LIN {X 0,Y 536.075,Z 1142.953,A -85,B 0,C 180,E1 24176.996,E2 24176.996} C_VEL
LIN {X 0,Y 540.442,Z 1123.188,A -85,B 0,C 180,E1 24174.545,E2 24174.545} C_VEL
LIN {X 0,Y 544.196,Z 1106.391,A -85,B 0,C 180,E1 24172.711,E2 24172.711} C_VEL
LIN {X 0,Y 547.982,Z 1089.375,A -85,B 0,C 180,E1 24171.05,E2 24171.05} C_VEL
LIN {X 0,Y 552.645,Z 1068.2,A -85,B 0,C 180,E1 24169.217,E2 24169.217} C_VEL
LIN {X 0,Y 557.206,Z 1046.015,A -85,B 0,C 180,E1 24167.564,E2 24167.564} C_VEL
LIN {X 0,Y 560.932,Z 1026.823,A -85,B 0,C 180,E1 24166.308,E2 24166.308} C_VEL
LIN {X 0,Y 564.507,Z 1007.094,A -85,B 0,C 180,E1 24165.17,E2 24165.17} C_VEL
LIN {X 0,Y 568.089,Z 985.711,A -85,B 0,C 180,E1 24164.098,E2 24164.098} C_VEL
LIN {X 0,Y 572.065,Z 959.057,A -85,B 0,C 180,E1 24162.974,E2 24162.974} C_VEL
LIN {X 0,Y 575.027,Z 935.232,A -85,B 0,C 180,E1 24162.158,E2 24162.158} C_VEL
LIN {X 0,Y 577.283,Z 914.135,A -85,B 0,C 180,E1 24161.567,E2 24161.567} C_VEL
LIN {X 0,Y 579.127,Z 892.797,A -85,B 0,C 180,E1 24161.086,E2 24161.086} C_VEL
LIN {X 0,Y 580.665,Z 868.419,A -85,B 0,C 180,E1 24160.665,E2 24160.665} C_VEL
LIN {X 0,Y 589.019,Z 647.142,A -85,B 0,C 180,E1 24157.424,E2 24157.424} C_VEL
LIN {X 0,Y 594.591,Z 507.254,A -85,B 0,C 180,E1 24155.344,E2 24155.344} C_VEL
LIN {X 0,Y 582.445,Z 490.253,A -85,B 0,C 180,E1 24153.234,E2 24153.234} C_VEL
LIN {X 0,Y 571.046,Z 475.195,A -85,B 0,C 180,E1 24151.071,E2 24151.071} C_VEL
LIN {X 0,Y 561.909,Z 463.769,A -85,B 0,C 180,E1 24149.181,E2 24149.181} C_VEL
LIN {X 0,Y 557.694,Z 458.589,A -85,B 0,C 180,E1 24148.251,E2 24148.251} C_VEL
LIN {X 0,Y 553.263,Z 453.23,A -85,B 0,C 180,E1 24147.227,E2 24147.227} C_VEL
LIN {X 0,Y 549.468,Z 448.48,A -85,B 0,C 180,E1 24146.302,E2 24146.302} C_VEL
LIN {X 0,Y 545.143,Z 443.711,A -85,B 0,C 180,E1 24145.213,E2 24145.213} C_VEL
LIN {X 0,Y 543.778,Z 441.838,A -85,B 0,C 180,E1 24144.845,E2 24144.845} C_VEL
LIN {X 0,Y 540.283,Z 438.305,A -85,B 0,C 180,E1 24143.91,E2 24143.91} C_VEL
LIN {X 0,Y 538.579,Z 435.768,A -85,B 0,C 180,E1 24143.41,E2 24143.41} C_VEL
LIN {X 0,Y 535.319,Z 432.979,A -85,B 0,C 180,E1 24142.485,E2 24142.485} C_VEL
LIN {X 0,Y 533.198,Z 429.458,A -85,B 0,C 180,E1 24141.796,E2 24141.796} C_VEL
LIN {X 0,Y 529.875,Z 427.069,A -85,B 0,C 180,E1 24140.779,E2 24140.779} C_VEL
LIN {X 0,Y 527.916,Z 423.816,A -85,B 0,C 180,E1 24140.078,E2 24140.078} C_VEL
LIN {X 0,Y 527.596,Z 422.918,A -85,B 0,C 180,E1 24139.946,E2 24139.946} C_VEL
LIN {X 0,Y 524.201,Z 421.053,A -85,B 0,C 180,E1 24138.806,E2 24138.806} C_VEL
LIN {X 0,Y 522.262,Z 418.242,A -85,B 0,C 180,E1 24138.04,E2 24138.04} C_VEL
LIN {X 0,Y 521.746,Z 416.24,A -85,B 0,C 180,E1 24137.731,E2 24137.731} C_VEL
LIN {X 0,Y 521.74,Z 416.177,A -85,B 0,C 180,E1 24134.2,E2 24134.2} C_VEL
LIN {X 0,Y 521.724,Z 416.212,A -85,B 0,C 180,E1 24130.826,E2 24130.826} C_VEL
LIN {X 0,Y 521.748,Z 416.194,A -85,B 0,C 180,E1 24127.267,E2 24127.267} C_VEL
LIN {X 0,Y 521.735,Z 416.182,A -85,B 0,C 180,E1 24123.846,E2 24123.846} C_VEL
LIN {X 0,Y 521.719,Z 416.225,A -85,B 0,C 180,E1 24120.439,E2 24120.439} C_VEL
LIN {X 0,Y 521.735,Z 416.172,A -85,B 0,C 180,E1 24117.034,E2 24117.034} C_VEL
LIN {X 0,Y 521.747,Z 416.238,A -85,B 0,C 180,E1 24113.508,E2 24113.508} C_VEL
LIN {X 0,Y 521.712,Z 416.179,A -85,B 0,C 180,E1 24110.067,E2 24110.067} C_VEL
LIN {X 0,Y 521.743,Z 416.199,A -85,B 0,C 180,E1 24106.592,E2 24106.592} C_VEL
LIN {X 0,Y 521.742,Z 416.215,A -85,B 0,C 180,E1 24103.064,E2 24103.064} C_VEL
LIN {X 0,Y 521.793,Z 416.552,A -85,B 0,C 180,E1 24102.836,E2 24102.836} C_VEL
LIN {X 0,Y 522.41,Z 418.598,A -85,B 0,C 180,E1 24102.311,E2 24102.311} C_VEL
LIN {X 0,Y 524.376,Z 421.238,A -85,B 0,C 180,E1 24101.547,E2 24101.547} C_VEL
LIN {X 0,Y 526.706,Z 422.973,A -85,B 0,C 180,E1 24100.741,E2 24100.741} C_VEL
LIN {X 0,Y 530.704,Z 427.887,A -85,B 0,C 180,E1 24099.37,E2 24099.37} C_VEL
LIN {X 0,Y 532.055,Z 429.416,A -85,B 0,C 180,E1 24098.936,E2 24098.936} C_VEL
LIN {X 0,Y 535.394,Z 433.498,A -85,B 0,C 180,E1 24097.894,E2 24097.894} C_VEL
LIN {X 0,Y 536.844,Z 435.07,A -85,B 0,C 180,E1 24097.467,E2 24097.467} C_VEL
LIN {X 0,Y 540.381,Z 439.58,A -85,B 0,C 180,E1 24096.442,E2 24096.442} C_VEL
LIN {X 0,Y 542.443,Z 442.092,A -85,B 0,C 180,E1 24095.873,E2 24095.873} C_VEL
LIN {X 0,Y 550.326,Z 451.99,A -85,B 0,C 180,E1 24093.832,E2 24093.832} C_VEL
LIN {X 0,Y 559.201,Z 463.612,A -85,B 0,C 180,E1 24091.745,E2 24091.745} C_VEL
LIN {X 0,Y 566.986,Z 474.312,A -85,B 0,C 180,E1 24090.061,E2 24090.061} C_VEL
LIN {X 0,Y 576.321,Z 487.386,A -85,B 0,C 180,E1 24088.197,E2 24088.197} C_VEL
LIN {X 0,Y 587.425,Z 503.948,A -85,B 0,C 180,E1 24086.149,E2 24086.149} C_VEL
LIN {X 0,Y 594.763,Z 515.576,A -85,B 0,C 180,E1 24084.879,E2 24084.879} C_VEL
LIN {X 0,Y 586.116,Z 737.329,A -85,B 0,C 180,E1 24081.599,E2 24081.599} C_VEL
LIN {X 0,Y 579.945,Z 901.421,A -85,B 0,C 180,E1 24079.193,E2 24079.193} C_VEL
LIN {X 0,Y 578.109,Z 926.813,A -85,B 0,C 180,E1 24078.724,E2 24078.724} C_VEL
LIN {X 0,Y 575.284,Z 954.698,A -85,B 0,C 180,E1 24078.019,E2 24078.019} C_VEL
LIN {X 0,Y 572.619,Z 976.547,A -85,B 0,C 180,E1 24077.322,E2 24077.322} C_VEL
LIN {X 0,Y 569.746,Z 997.313,A -85,B 0,C 180,E1 24076.532,E2 24076.532} C_VEL
LIN {X 0,Y 566.591,Z 1017.778,A -85,B 0,C 180,E1 24075.624,E2 24075.624} C_VEL
LIN {X 0,Y 562.4,Z 1042.853,A -85,B 0,C 180,E1 24074.327,E2 24074.327} C_VEL
LIN {X 0,Y 557.928,Z 1066.671,A -85,B 0,C 180,E1 24072.862,E2 24072.862} C_VEL
LIN {X 0,Y 554.11,Z 1086.01,A -85,B 0,C 180,E1 24071.507,E2 24071.507} C_VEL
LIN {X 0,Y 550.291,Z 1104.678,A -85,B 0,C 180,E1 24070.036,E2 24070.036} C_VEL
LIN {X 0,Y 545.836,Z 1126.18,A -85,B 0,C 180,E1 24068.125,E2 24068.125} C_VEL
LIN {X 0,Y 541.315,Z 1147.112,A -85,B 0,C 180,E1 24065.976,E2 24065.976} C_VEL
LIN {X 0,Y 537.945,Z 1162.95,A -85,B 0,C 180,E1 24064.152,E2 24064.152} C_VEL
LIN {X 0,Y 534.756,Z 1178.185,A -85,B 0,C 180,E1 24062.205,E2 24062.205} C_VEL
LIN {X 0,Y 531.96,Z 1191.879,A -85,B 0,C 180,E1 24060.252,E2 24060.252} C_VEL
LIN {X 0,Y 528.767,Z 1208.247,A -85,B 0,C 180,E1 24057.603,E2 24057.603} C_VEL
LIN {X 0,Y 526.236,Z 1221.814,A -85,B 0,C 180,E1 24055.073,E2 24055.073} C_VEL
LIN {X 0,Y 524.432,Z 1232.748,A -85,B 0,C 180,E1 24052.775,E2 24052.775} C_VEL
LIN {X 0,Y 522.972,Z 1242.875,A -85,B 0,C 180,E1 24050.367,E2 24050.367} C_VEL
LIN {X 0,Y 521.584,Z 1254.016,A -85,B 0,C 180,E1 24047.29,E2 24047.29} C_VEL
LIN {X 0,Y 520.805,Z 1261.822,A -85,B 0,C 180,E1 24044.685,E2 24044.685} C_VEL
LIN {X 0,Y 520.372,Z 1267.788,A -85,B 0,C 180,E1 24042.319,E2 24042.319} C_VEL
LIN {X 0,Y 520.094,Z 1272.687,A -85,B 0,C 180,E1 24039.968,E2 24039.968} C_VEL
LIN {X 0,Y 519.963,Z 1276.513,A -85,B 0,C 180,E1 24037.63,E2 24037.63} C_VEL
LIN {X 0,Y 519.924,Z 1279.425,A -85,B 0,C 180,E1 24035.191,E2 24035.191} C_VEL
LIN {X 0,Y 519.907,Z 1281.486,A -85,B 0,C 180,E1 24032.32,E2 24032.32} C_VEL
LIN {X 0,Y 519.867,Z 1281.895,A -85,B 0,C 180,E1 24029.454,E2 24029.454} C_VEL
LIN {X 0,Y 519.91,Z 1281.085,A -85,B 0,C 180,E1 24027.029,E2 24027.029} C_VEL
LIN {X 0,Y 519.927,Z 1279.207,A -85,B 0,C 180,E1 24024.598,E2 24024.598} C_VEL
LIN {X 0,Y 519.965,Z 1276.367,A -85,B 0,C 180,E1 24022.269,E2 24022.269} C_VEL
LIN {X 0,Y 520.127,Z 1272.292,A -85,B 0,C 180,E1 24019.819,E2 24019.819} C_VEL
LIN {X 0,Y 520.466,Z 1266.539,A -85,B 0,C 180,E1 24017.129,E2 24017.129} C_VEL
LIN {X 0,Y 521.147,Z 1258.286,A -85,B 0,C 180,E1 24014.082,E2 24014.082} C_VEL
LIN {X 0,Y 522.031,Z 1250.124,A -85,B 0,C 180,E1 24011.583,E2 24011.583} C_VEL
LIN {X 0,Y 523.22,Z 1241.086,A -85,B 0,C 180,E1 24009.186,E2 24009.186} C_VEL
LIN {X 0,Y 524.855,Z 1230.228,A -85,B 0,C 180,E1 24006.663,E2 24006.663} C_VEL
LIN {X 0,Y 527.434,Z 1215.294,A -85,B 0,C 180,E1 24003.673,E2 24003.673} C_VEL
LIN {X 0,Y 529.89,Z 1202.104,A -85,B 0,C 180,E1 24001.368,E2 24001.368} C_VEL
LIN {X 0,Y 532.584,Z 1188.867,A -85,B 0,C 180,E1 23999.3,E2 23999.3} C_VEL
LIN {X 0,Y 535.438,Z 1175.023,A -85,B 0,C 180,E1 23997.374,E2 23997.374} C_VEL
LIN {X 0,Y 539.472,Z 1155.985,A -85,B 0,C 180,E1 23995.008,E2 23995.008} C_VEL
LIN {X 0,Y 543.566,Z 1136.456,A -85,B 0,C 180,E1 23992.898,E2 23992.898} C_VEL
LIN {X 0,Y 547.292,Z 1118.896,A -85,B 0,C 180,E1 23991.205,E2 23991.205} C_VEL
LIN {X 0,Y 551.093,Z 1100.741,A -85,B 0,C 180,E1 23989.638,E2 23989.638} C_VEL
LIN {X 0,Y 555.864,Z 1077.535,A -85,B 0,C 180,E1 23987.869,E2 23987.869} C_VEL
LIN {X 0,Y 560.167,Z 1054.848,A -85,B 0,C 180,E1 23986.388,E2 23986.388} C_VEL
LIN {X 0,Y 563.715,Z 1034.948,A -85,B 0,C 180,E1 23985.247,E2 23985.247} C_VEL
LIN {X 0,Y 567.094,Z 1014.57,A -85,B 0,C 180,E1 23984.225,E2 23984.225} C_VEL
LIN {X 0,Y 570.382,Z 992.949,A -85,B 0,C 180,E1 23983.29,E2 23983.29} C_VEL
LIN {X 0,Y 574.097,Z 964.972,A -85,B 0,C 180,E1 23982.289,E2 23982.289} C_VEL
LIN {X 0,Y 576.725,Z 941.016,A -85,B 0,C 180,E1 23981.613,E2 23981.613} C_VEL
LIN {X 0,Y 578.683,Z 919.422,A -85,B 0,C 180,E1 23981.129,E2 23981.129} C_VEL
LIN {X 0,Y 580.174,Z 896.923,A -85,B 0,C 180,E1 23980.736,E2 23980.736} C_VEL
LIN {X 0,Y 588.374,Z 677.174,A -85,B 0,C 180,E1 23977.519,E2 23977.519} C_VEL
LIN {X 0,Y 594.647,Z 515.244,A -85,B 0,C 180,E1 23975.105,E2 23975.105} C_VEL
LIN {X 0,Y 583.42,Z 497.942,A -85,B 0,C 180,E1 23973.142,E2 23973.142} C_VEL
LIN {X 0,Y 572.285,Z 481.584,A -85,B 0,C 180,E1 23971.026,E2 23971.026} C_VEL
LIN {X 0,Y 561.441,Z 466.668,A -85,B 0,C 180,E1 23968.77,E2 23968.77} C_VEL
LIN {X 0,Y 553.204,Z 455.818,A -85,B 0,C 180,E1 23966.892,E2 23966.892} C_VEL
LIN {X 0,Y 547.92,Z 449.108,A -85,B 0,C 180,E1 23965.597,E2 23965.597} C_VEL
LIN {X 0,Y 544.163,Z 444.377,A -85,B 0,C 180,E1 23964.623,E2 23964.623} C_VEL
LIN {X 0,Y 540.459,Z 439.692,A -85,B 0,C 180,E1 23963.612,E2 23963.612} C_VEL
LIN {X 0,Y 536.737,Z 434.957,A -85,B 0,C 180,E1 23962.538,E2 23962.538} C_VEL
LIN {X 0,Y 532.325,Z 429.897,A -85,B 0,C 180,E1 23961.197,E2 23961.197} C_VEL
LIN {X 0,Y 531.065,Z 428.242,A -85,B 0,C 180,E1 23960.788,E2 23960.788} C_VEL
LIN {X 0,Y 526.86,Z 423.282,A -85,B 0,C 180,E1 23959.369,E2 23959.369} C_VEL
LIN {X 0,Y 526.049,Z 422.369,A -85,B 0,C 180,E1 23959.083,E2 23959.083} C_VEL
LIN {X 0,Y 523.247,Z 420.086,A -85,B 0,C 180,E1 23958.091,E2 23958.091} C_VEL
LIN {X 0,Y 521.979,Z 417.463,A -85,B 0,C 180,E1 23957.482,E2 23957.482} C_VEL
LIN {X 0,Y 521.684,Z 416.232,A -85,B 0,C 180,E1 23957.053,E2 23957.053} C_VEL
LIN {X 0,Y 521.665,Z 416.192,A -85,B 0,C 180,E1 23953.976,E2 23953.976} C_VEL
LIN {X 0,Y 521.65,Z 416.207,A -85,B 0,C 180,E1 23950.604,E2 23950.604} C_VEL
LIN {X 0,Y 521.72,Z 416.209,A -85,B 0,C 180,E1 23947.267,E2 23947.267} C_VEL
LIN {X 0,Y 521.646,Z 416.191,A -85,B 0,C 180,E1 23943.957,E2 23943.957} C_VEL
LIN {X 0,Y 521.666,Z 416.246,A -85,B 0,C 180,E1 23940.439,E2 23940.439} C_VEL
LIN {X 0,Y 521.695,Z 416.178,A -85,B 0,C 180,E1 23937.254,E2 23937.254} C_VEL
LIN {X 0,Y 521.667,Z 416.251,A -85,B 0,C 180,E1 23933.949,E2 23933.949} C_VEL
LIN {X 0,Y 521.724,Z 416.175,A -85,B 0,C 180,E1 23930.701,E2 23930.701} C_VEL
LIN {X 0,Y 521.686,Z 416.234,A -85,B 0,C 180,E1 23927.379,E2 23927.379} C_VEL
LIN {X 0,Y 521.681,Z 416.196,A -85,B 0,C 180,E1 23923.864,E2 23923.864} C_VEL
LIN {X 0,Y 521.734,Z 416.445,A -85,B 0,C 180,E1 23922.071,E2 23922.071} C_VEL
LIN {X 0,Y 522.615,Z 419.098,A -85,B 0,C 180,E1 23921.655,E2 23921.655} C_VEL
LIN {X 0,Y 524.863,Z 421.607,A -85,B 0,C 180,E1 23920.815,E2 23920.815} C_VEL
LIN {X 0,Y 527.594,Z 423.099,A -85,B 0,C 180,E1 23919.909,E2 23919.909} C_VEL
LIN {X 0,Y 529.36,Z 426.472,A -85,B 0,C 180,E1 23919.258,E2 23919.258} C_VEL
LIN {X 0,Y 532.458,Z 429.11,A -85,B 0,C 180,E1 23918.288,E2 23918.288} C_VEL
LIN {X 0,Y 533.39,Z 429.812,A -85,B 0,C 180,E1 23918.01,E2 23918.01} C_VEL
LIN {X 0,Y 535.705,Z 433.45,A -85,B 0,C 180,E1 23917.271,E2 23917.271} C_VEL
LIN {X 0,Y 538.99,Z 436.275,A -85,B 0,C 180,E1 23916.349,E2 23916.349} C_VEL
LIN {X 0,Y 541.875,Z 440.251,A -85,B 0,C 180,E1 23915.527,E2 23915.527} C_VEL
LIN {X 0,Y 544.409,Z 442.624,A -85,B 0,C 180,E1 23914.868,E2 23914.868} C_VEL
LIN {X 0,Y 547.687,Z 446.838,A -85,B 0,C 180,E1 23914.013,E2 23914.013} C_VEL
LIN {X 0,Y 549.655,Z 448.85,A -85,B 0,C 180,E1 23913.533,E2 23913.533} C_VEL
LIN {X 0,Y 553.418,Z 453.418,A -85,B 0,C 180,E1 23912.624,E2 23912.624} C_VEL
LIN {X 0,Y 559.71,Z 461.077,A -85,B 0,C 180,E1 23911.191,E2 23911.191} C_VEL
LIN {X 0,Y 565.074,Z 467.811,A -85,B 0,C 180,E1 23910.037,E2 23910.037} C_VEL
LIN {X 0,Y 572.456,Z 477.096,A -85,B 0,C 180,E1 23908.546,E2 23908.546} C_VEL
LIN {X 0,Y 583.839,Z 492.189,A -85,B 0,C 180,E1 23906.415,E2 23906.415} C_VEL
LIN {X 0,Y 594.576,Z 507.251,A -85,B 0,C 180,E1 23904.562,E2 23904.562} C_VEL
LIN {X 0,Y 586.202,Z 720.061,A -85,B 0,C 180,E1 23901.412,E2 23901.412} C_VEL
LIN {X 0,Y 580.222,Z 876.564,A -85,B 0,C 180,E1 23899.114,E2 23899.114} C_VEL
LIN {X 0,Y 578.508,Z 900.954,A -85,B 0,C 180,E1 23898.656,E2 23898.656} C_VEL
LIN {X 0,Y 575.746,Z 929.049,A -85,B 0,C 180,E1 23897.938,E2 23897.938} C_VEL
LIN {X 0,Y 573.071,Z 951.13,A -85,B 0,C 180,E1 23897.223,E2 23897.223} C_VEL
LIN {X 0,Y 572.664,Z 954.299,A -85,B 0,C 180,E1 23897.108,E2 23897.108} C_VEL
LIN {X 0,Y 571.028,Z 961.789,A -85,B 0,C 180,E1 23896.911,E2 23896.911} C_VEL
LIN {X 0,Y 564.119,Z 980.351,A -85,B 0,C 180,E1 23896.593,E2 23896.593} C_VEL
LIN {X 0,Y 562.235,Z 987.347,A -85,B 0,C 180,E1 23896.34,E2 23896.34} C_VEL
LIN {X 0,Y 558.591,Z 1008.291,A -85,B 0,C 180,E1 23895.277,E2 23895.277} C_VEL
LIN {X 0,Y 554.89,Z 1027.907,A -85,B 0,C 180,E1 23894.134,E2 23894.134} C_VEL
LIN {X 0,Y 550.282,Z 1050.7,A -85,B 0,C 180,E1 23892.616,E2 23892.616} C_VEL
LIN {X 0,Y 545.35,Z 1072.999,A -85,B 0,C 180,E1 23890.877,E2 23890.877} C_VEL
LIN {X 0,Y 541.243,Z 1091.032,A -85,B 0,C 180,E1 23889.28,E2 23889.28} C_VEL
LIN {X 0,Y 537.325,Z 1107.891,A -85,B 0,C 180,E1 23887.607,E2 23887.607} C_VEL
LIN {X 0,Y 532.822,Z 1127.36,A -85,B 0,C 180,E1 23885.433,E2 23885.433} C_VEL
LIN {X 0,Y 528.487,Z 1145.755,A -85,B 0,C 180,E1 23883.054,E2 23883.054} C_VEL
LIN {X 0,Y 525.317,Z 1159.609,A -85,B 0,C 180,E1 23881.045,E2 23881.045} C_VEL
LIN {X 0,Y 522.449,Z 1172.564,A -85,B 0,C 180,E1 23878.953,E2 23878.953} C_VEL
LIN {X 0,Y 519.628,Z 1186.965,A -85,B 0,C 180,E1 23876.384,E2 23876.384} C_VEL
LIN {X 0,Y 517.048,Z 1201.064,A -85,B 0,C 180,E1 23873.469,E2 23873.469} C_VEL
LIN {X 0,Y 515.412,Z 1211.37,A -85,B 0,C 180,E1 23871.026,E2 23871.026} C_VEL
LIN {X 0,Y 514.151,Z 1220.373,A -85,B 0,C 180,E1 23868.592,E2 23868.592} C_VEL
LIN {X 0,Y 513.107,Z 1229.901,A -85,B 0,C 180,E1 23865.594,E2 23865.594} C_VEL
LIN {X 0,Y 512.44,Z 1237.323,A -85,B 0,C 180,E1 23862.677,E2 23862.677} C_VEL
LIN {X 0,Y 512.144,Z 1242.414,A -85,B 0,C 180,E1 23860.228,E2 23860.228} C_VEL
LIN {X 0,Y 511.965,Z 1246.46,A -85,B 0,C 180,E1 23857.739,E2 23857.739} C_VEL
LIN {X 0,Y 511.926,Z 1249.386,A -85,B 0,C 180,E1 23855.262,E2 23855.262} C_VEL
LIN {X 0,Y 511.909,Z 1251.397,A -85,B 0,C 180,E1 23852.458,E2 23852.458} C_VEL
LIN {X 0,Y 511.869,Z 1251.902,A -85,B 0,C 180,E1 23849.435,E2 23849.435} C_VEL
LIN {X 0,Y 511.909,Z 1251.106,A -85,B 0,C 180,E1 23846.972,E2 23846.972} C_VEL
LIN {X 0,Y 511.928,Z 1249.24,A -85,B 0,C 180,E1 23844.503,E2 23844.503} C_VEL
LIN {X 0,Y 511.973,Z 1246.414,A -85,B 0,C 180,E1 23842.138,E2 23842.138} C_VEL
LIN {X 0,Y 512.15,Z 1242.352,A -85,B 0,C 180,E1 23839.648,E2 23839.648} C_VEL
LIN {X 0,Y 512.512,Z 1236.616,A -85,B 0,C 180,E1 23836.916,E2 23836.916} C_VEL
LIN {X 0,Y 513.228,Z 1228.392,A -85,B 0,C 180,E1 23833.819,E2 23833.819} C_VEL
LIN {X 0,Y 514.167,Z 1220.22,A -85,B 0,C 180,E1 23831.274,E2 23831.274} C_VEL
LIN {X 0,Y 515.43,Z 1211.212,A -85,B 0,C 180,E1 23828.845,E2 23828.845} C_VEL
LIN {X 0,Y 517.083,Z 1200.879,A -85,B 0,C 180,E1 23826.4,E2 23826.4} C_VEL
LIN {X 0,Y 519.684,Z 1186.642,A -85,B 0,C 180,E1 23823.467,E2 23823.467} C_VEL
LIN {X 0,Y 522.504,Z 1172.306,A -85,B 0,C 180,E1 23820.914,E2 23820.914} C_VEL
LIN {X 0,Y 525.384,Z 1159.319,A -85,B 0,C 180,E1 23818.821,E2 23818.821} C_VEL
LIN {X 0,Y 528.746,Z 1144.669,A -85,B 0,C 180,E1 23816.705,E2 23816.705} C_VEL
LIN {X 0,Y 533.455,Z 1124.453,A -85,B 0,C 180,E1 23814.141,E2 23814.141} C_VEL
LIN {X 0,Y 537.444,Z 1107.389,A -85,B 0,C 180,E1 23812.251,E2 23812.251} C_VEL
LIN {X 0,Y 541.29,Z 1090.841,A -85,B 0,C 180,E1 23810.612,E2 23810.612} C_VEL
LIN {X 0,Y 545.246,Z 1073.473,A -85,B 0,C 180,E1 23809.073,E2 23809.073} C_VEL
LIN {X 0,Y 550.207,Z 1051.088,A -85,B 0,C 180,E1 23807.321,E2 23807.321} C_VEL
LIN {X 0,Y 554.881,Z 1027.974,A -85,B 0,C 180,E1 23805.78,E2 23805.78} C_VEL
LIN {X 0,Y 558.581,Z 1008.349,A -85,B 0,C 180,E1 23804.636,E2 23804.636} C_VEL
LIN {X 0,Y 562.092,Z 988.212,A -85,B 0,C 180,E1 23803.611,E2 23803.611} C_VEL
LIN {X 0,Y 565.567,Z 966.271,A -85,B 0,C 180,E1 23802.65,E2 23802.65} C_VEL
LIN {X 0,Y 569.342,Z 938.225,A -85,B 0,C 180,E1 23801.642,E2 23801.642} C_VEL
LIN {X 0,Y 571.853,Z 915.757,A -85,B 0,C 180,E1 23801.001,E2 23801.001} C_VEL
LIN {X 0,Y 573.785,Z 894.335,A -85,B 0,C 180,E1 23800.509,E2 23800.509} C_VEL
LIN {X 0,Y 575.294,Z 871.966,A -85,B 0,C 180,E1 23800.113,E2 23800.113} C_VEL
LIN {X 0,Y 583.962,Z 652.814,A -85,B 0,C 180,E1 23796.88,E2 23796.88} C_VEL
LIN {X 0,Y 589.757,Z 511.444,A -85,B 0,C 180,E1 23794.76,E2 23794.76} C_VEL
LIN {X 0,Y 578.023,Z 495.117,A -85,B 0,C 180,E1 23792.664,E2 23792.664} C_VEL
LIN {X 0,Y 568.051,Z 481.818,A -85,B 0,C 180,E1 23790.724,E2 23790.724} C_VEL
LIN {X 0,Y 559.134,Z 470.542,A -85,B 0,C 180,E1 23788.842,E2 23788.842} C_VEL
LIN {X 0,Y 555.074,Z 465.514,A -85,B 0,C 180,E1 23787.928,E2 23787.928} C_VEL
LIN {X 0,Y 550.733,Z 460.238,A -85,B 0,C 180,E1 23786.906,E2 23786.906} C_VEL
LIN {X 0,Y 546.167,Z 454.703,A -85,B 0,C 180,E1 23785.773,E2 23785.773} C_VEL
LIN {X 0,Y 542.432,Z 450.174,A -85,B 0,C 180,E1 23784.794,E2 23784.794} C_VEL
LIN {X 0,Y 537.827,Z 445.071,A -85,B 0,C 180,E1 23783.531,E2 23783.531} C_VEL
LIN {X 0,Y 536.56,Z 443.245,A -85,B 0,C 180,E1 23783.154,E2 23783.154} C_VEL
LIN {X 0,Y 533.107,Z 440.023,A -85,B 0,C 180,E1 23782.148,E2 23782.148} C_VEL
LIN {X 0,Y 531.239,Z 437.012,A -85,B 0,C 180,E1 23781.532,E2 23781.532} C_VEL
LIN {X 0,Y 527.981,Z 434.437,A -85,B 0,C 180,E1 23780.509,E2 23780.509} C_VEL
LIN {X 0,Y 525.704,Z 430.592,A -85,B 0,C 180,E1 23779.673,E2 23779.673} C_VEL
LIN {X 0,Y 522.389,Z 428.464,A -85,B 0,C 180,E1 23778.526,E2 23778.526} C_VEL
LIN {X 0,Y 520.305,Z 425.264,A -85,B 0,C 180,E1 23777.676,E2 23777.676} C_VEL
LIN {X 0,Y 519.854,Z 424.016,A -85,B 0,C 180,E1 23777.461,E2 23777.461} C_VEL
LIN {X 0,Y 516.371,Z 422.127,A -85,B 0,C 180,E1 23776.076,E2 23776.076} C_VEL
LIN {X 0,Y 514.326,Z 419.231,A -85,B 0,C 180,E1 23775.1,E2 23775.1} C_VEL
LIN {X 0,Y 513.784,Z 417.163,A -85,B 0,C 180,E1 23774.737,E2 23774.737} C_VEL
LIN {X 0,Y 513.796,Z 417.213,A -85,B 0,C 180,E1 23771.222,E2 23771.222} C_VEL
LIN {X 0,Y 513.797,Z 417.17,A -85,B 0,C 180,E1 23767.717,E2 23767.717} C_VEL
LIN {X 0,Y 513.782,Z 417.183,A -85,B 0,C 180,E1 23764.353,E2 23764.353} C_VEL
LIN {X 0,Y 513.789,Z 417.195,A -85,B 0,C 180,E1 23760.781,E2 23760.781} C_VEL
LIN {X 0,Y 513.796,Z 417.163,A -85,B 0,C 180,E1 23757.435,E2 23757.435} C_VEL
LIN {X 0,Y 513.785,Z 417.227,A -85,B 0,C 180,E1 23753.968,E2 23753.968} C_VEL
LIN {X 0,Y 513.786,Z 417.161,A -85,B 0,C 180,E1 23750.478,E2 23750.478} C_VEL
LIN {X 0,Y 513.805,Z 417.201,A -85,B 0,C 180,E1 23747.068,E2 23747.068} C_VEL
LIN {X 0,Y 513.811,Z 417.4,A -85,B 0,C 180,E1 23745.634,E2 23745.634} C_VEL
LIN {X 0,Y 514.771,Z 420.1,A -85,B 0,C 180,E1 23745.086,E2 23745.086} C_VEL
LIN {X 0,Y 517.285,Z 422.855,A -85,B 0,C 180,E1 23743.954,E2 23743.954} C_VEL
LIN {X 0,Y 519.713,Z 424.242,A -85,B 0,C 180,E1 23742.996,E2 23742.996} C_VEL
LIN {X 0,Y 522.136,Z 428.235,A -85,B 0,C 180,E1 23741.985,E2 23741.985} C_VEL
LIN {X 0,Y 525.064,Z 430.697,A -85,B 0,C 180,E1 23740.938,E2 23740.938} C_VEL
LIN {X 0,Y 529.434,Z 435.843,A -85,B 0,C 180,E1 23739.434,E2 23739.434} C_VEL
LIN {X 0,Y 533.42,Z 440.887,A -85,B 0,C 180,E1 23738.156,E2 23738.156} C_VEL
LIN {X 0,Y 535.01,Z 442.752,A -85,B 0,C 180,E1 23737.675,E2 23737.675} C_VEL
LIN {X 0,Y 538.891,Z 447.461,A -85,B 0,C 180,E1 23736.547,E2 23736.547} C_VEL
LIN {X 0,Y 548.186,Z 459.455,A -85,B 0,C 180,E1 23734.068,E2 23734.068} C_VEL
LIN {X 0,Y 556.559,Z 470.49,A -85,B 0,C 180,E1 23732.066,E2 23732.066} C_VEL
LIN {X 0,Y 564.579,Z 481.644,A -85,B 0,C 180,E1 23730.301,E2 23730.301} C_VEL
LIN {X 0,Y 573.533,Z 494.355,A -85,B 0,C 180,E1 23728.483,E2 23728.483} C_VEL
LIN {X 0,Y 584.362,Z 510.722,A -85,B 0,C 180,E1 23726.449,E2 23726.449} C_VEL
LIN {X 0,Y 589.973,Z 519.666,A -85,B 0,C 180,E1 23725.455,E2 23725.455} C_VEL
LIN {X 0,Y 581.03,Z 740.052,A -85,B 0,C 180,E1 23722.178,E2 23722.178} C_VEL
LIN {X 0,Y 574.716,Z 901.172,A -85,B 0,C 180,E1 23719.801,E2 23719.801} C_VEL
LIN {X 0,Y 572.793,Z 926.885,A -85,B 0,C 180,E1 23719.324,E2 23719.324} C_VEL
LIN {X 0,Y 569.871,Z 954.622,A -85,B 0,C 180,E1 23718.62,E2 23718.62} C_VEL
LIN {X 0,Y 567.136,Z 976.287,A -85,B 0,C 180,E1 23717.926,E2 23717.926} C_VEL
LIN {X 0,Y 564.233,Z 996.519,A -85,B 0,C 180,E1 23717.156,E2 23717.156} C_VEL
LIN {X 0,Y 561.04,Z 1016.488,A -85,B 0,C 180,E1 23716.272,E2 23716.272} C_VEL
LIN {X 0,Y 557.204,Z 1038.542,A -85,B 0,C 180,E1 23715.142,E2 23715.142} C_VEL
LIN {X 0,Y 552.193,Z 1064.748,A -85,B 0,C 180,E1 23713.561,E2 23713.561} C_VEL
LIN {X 0,Y 548.114,Z 1084.598,A -85,B 0,C 180,E1 23712.172,E2 23712.172} C_VEL
LIN {X 0,Y 544.181,Z 1103.052,A -85,B 0,C 180,E1 23710.718,E2 23710.718} C_VEL
LIN {X 0,Y 540.121,Z 1121.591,A -85,B 0,C 180,E1 23709.079,E2 23709.079} C_VEL
LIN {X 0,Y 535.235,Z 1143.751,A -85,B 0,C 180,E1 23706.85,E2 23706.85} C_VEL
LIN {X 0,Y 531.185,Z 1161.733,A -85,B 0,C 180,E1 23704.779,E2 23704.779} C_VEL
LIN {X 0,Y 527.826,Z 1177.049,A -85,B 0,C 180,E1 23702.809,E2 23702.809} C_VEL
LIN {X 0,Y 524.69,Z 1191.694,A -85,B 0,C 180,E1 23700.716,E2 23700.716} C_VEL
LIN {X 0,Y 521.429,Z 1207.849,A -85,B 0,C 180,E1 23698.103,E2 23698.103} C_VEL
LIN {X 0,Y 518.667,Z 1221.812,A -85,B 0,C 180,E1 23695.465,E2 23695.465} C_VEL
LIN {X 0,Y 516.755,Z 1232.746,A -85,B 0,C 180,E1 23693.132,E2 23693.132} C_VEL
LIN {X 0,Y 515.195,Z 1242.874,A -85,B 0,C 180,E1 23690.689,E2 23690.689} C_VEL
LIN {X 0,Y 513.756,Z 1253.66,A -85,B 0,C 180,E1 23687.679,E2 23687.679} C_VEL
LIN {X 0,Y 512.89,Z 1261.821,A -85,B 0,C 180,E1 23684.916,E2 23684.916} C_VEL
LIN {X 0,Y 512.408,Z 1267.788,A -85,B 0,C 180,E1 23682.514,E2 23682.514} C_VEL
LIN {X 0,Y 512.122,Z 1272.684,A -85,B 0,C 180,E1 23680.125,E2 23680.125} C_VEL
LIN {X 0,Y 511.965,Z 1276.67,A -85,B 0,C 180,E1 23677.637,E2 23677.637} C_VEL
LIN {X 0,Y 511.925,Z 1279.658,A -85,B 0,C 180,E1 23675.038,E2 23675.038} C_VEL
LIN {X 0,Y 511.91,Z 1281.598,A -85,B 0,C 180,E1 23672.02,E2 23672.02} C_VEL
LIN {X 0,Y 511.865,Z 1281.872,A -85,B 0,C 180,E1 23669.334,E2 23669.334} C_VEL
LIN {X 0,Y 511.91,Z 1281.085,A -85,B 0,C 180,E1 23666.982,E2 23666.982} C_VEL
LIN {X 0,Y 511.93,Z 1279.204,A -85,B 0,C 180,E1 23664.514,E2 23664.514} C_VEL
LIN {X 0,Y 511.97,Z 1276.364,A -85,B 0,C 180,E1 23662.148,E2 23662.148} C_VEL
LIN {X 0,Y 512.155,Z 1272.289,A -85,B 0,C 180,E1 23659.659,E2 23659.659} C_VEL
LIN {X 0,Y 512.542,Z 1266.284,A -85,B 0,C 180,E1 23656.812,E2 23656.812} C_VEL
LIN {X 0,Y 513.276,Z 1257.932,A -85,B 0,C 180,E1 23653.715,E2 23653.715} C_VEL
LIN {X 0,Y 514.226,Z 1249.718,A -85,B 0,C 180,E1 23651.175,E2 23651.175} C_VEL
LIN {X 0,Y 515.452,Z 1241.084,A -85,B 0,C 180,E1 23648.857,E2 23648.857} C_VEL
LIN {X 0,Y 517.11,Z 1230.741,A -85,B 0,C 180,E1 23646.413,E2 23646.413} C_VEL
LIN {X 0,Y 519.813,Z 1215.927,A -85,B 0,C 180,E1 23643.38,E2 23643.38} C_VEL
LIN {X 0,Y 522.445,Z 1202.555,A -85,B 0,C 180,E1 23641.003,E2 23641.003} C_VEL
LIN {X 0,Y 525.177,Z 1189.415,A -85,B 0,C 180,E1 23638.946,E2 23638.946} C_VEL
LIN {X 0,Y 528.19,Z 1175.41,A -85,B 0,C 180,E1 23636.97,E2 23636.97} C_VEL
LIN {X 0,Y 532.137,Z 1157.59,A -85,B 0,C 180,E1 23634.713,E2 23634.713} C_VEL
LIN {X 0,Y 536.746,Z 1136.742,A -85,B 0,C 180,E1 23632.413,E2 23632.413} C_VEL
LIN {X 0,Y 540.636,Z 1119.237,A -85,B 0,C 180,E1 23630.704,E2 23630.704} C_VEL
LIN {X 0,Y 544.594,Z 1101.142,A -85,B 0,C 180,E1 23629.124,E2 23629.124} C_VEL
LIN {X 0,Y 549.223,Z 1079.529,A -85,B 0,C 180,E1 23627.452,E2 23627.452} C_VEL
LIN {X 0,Y 554.031,Z 1055.482,A -85,B 0,C 180,E1 23625.852,E2 23625.852} C_VEL
LIN {X 0,Y 557.712,Z 1035.688,A -85,B 0,C 180,E1 23624.705,E2 23624.705} C_VEL
LIN {X 0,Y 561.21,Z 1015.434,A -85,B 0,C 180,E1 23623.678,E2 23623.678} C_VEL
LIN {X 0,Y 564.495,Z 994.73,A -85,B 0,C 180,E1 23622.771,E2 23622.771} C_VEL
LIN {X 0,Y 567.928,Z 970.58,A -85,B 0,C 180,E1 23621.875,E2 23621.875} C_VEL
LIN {X 0,Y 571.183,Z 942.806,A -85,B 0,C 180,E1 23621.059,E2 23621.059} C_VEL
LIN {X 0,Y 573.305,Z 920.449,A -85,B 0,C 180,E1 23620.548,E2 23620.548} C_VEL
LIN {X 0,Y 574.868,Z 898.147,A -85,B 0,C 180,E1 23620.152,E2 23620.152} C_VEL
LIN {X 0,Y 583.325,Z 681.23,A -85,B 0,C 180,E1 23616.955,E2 23616.955} C_VEL
LIN {X 0,Y 589.902,Z 519.357,A -85,B 0,C 180,E1 23614.536,E2 23614.536} C_VEL
LIN {X 0,Y 578.288,Z 501.441,A -85,B 0,C 180,E1 23612.442,E2 23612.442} C_VEL
LIN {X 0,Y 566.168,Z 483.765,A -85,B 0,C 180,E1 23610.045,E2 23610.045} C_VEL
LIN {X 0,Y 555.258,Z 468.753,A -85,B 0,C 180,E1 23607.655,E2 23607.655} C_VEL
LIN {X 0,Y 545.993,Z 456.694,A -85,B 0,C 180,E1 23605.403,E2 23605.403} C_VEL
LIN {X 0,Y 538.602,Z 447.234,A -85,B 0,C 180,E1 23603.408,E2 23603.408} C_VEL
LIN {X 0,Y 534.74,Z 442.368,A -85,B 0,C 180,E1 23602.279,E2 23602.279} C_VEL
LIN {X 0,Y 530.236,Z 437.036,A -85,B 0,C 180,E1 23600.88,E2 23600.88} C_VEL
LIN {X 0,Y 528.661,Z 435.236,A -85,B 0,C 180,E1 23600.366,E2 23600.366} C_VEL
LIN {X 0,Y 524.493,Z 430.094,A -85,B 0,C 180,E1 23598.91,E2 23598.91} C_VEL
LIN {X 0,Y 521.584,Z 427.63,A -85,B 0,C 180,E1 23597.862,E2 23597.862} C_VEL
LIN {X 0,Y 519.299,Z 423.867,A -85,B 0,C 180,E1 23596.903,E2 23596.903} C_VEL
LIN {X 0,Y 516.119,Z 421.909,A -85,B 0,C 180,E1 23595.622,E2 23595.622} C_VEL
LIN {X 0,Y 514.195,Z 419.077,A -85,B 0,C 180,E1 23594.701,E2 23594.701} C_VEL
LIN {X 0,Y 513.709,Z 417.176,A -85,B 0,C 180,E1 23594.369,E2 23594.369} C_VEL
LIN {X 0,Y 513.742,Z 417.202,A -85,B 0,C 180,E1 23590.996,E2 23590.996} C_VEL
LIN {X 0,Y 513.724,Z 417.188,A -85,B 0,C 180,E1 23587.718,E2 23587.718} C_VEL
LIN {X 0,Y 513.707,Z 417.185,A -85,B 0,C 180,E1 23584.354,E2 23584.354} C_VEL
LIN {X 0,Y 513.782,Z 417.204,A -85,B 0,C 180,E1 23581.004,E2 23581.004} C_VEL
LIN {X 0,Y 513.717,Z 417.174,A -85,B 0,C 180,E1 23577.769,E2 23577.769} C_VEL
LIN {X 0,Y 513.736,Z 417.238,A -85,B 0,C 180,E1 23574.191,E2 23574.191} C_VEL
LIN {X 0,Y 513.772,Z 417.163,A -85,B 0,C 180,E1 23571.043,E2 23571.043} C_VEL
LIN {X 0,Y 513.739,Z 417.232,A -85,B 0,C 180,E1 23567.638,E2 23567.638} C_VEL
LIN {X 0,Y 513.788,Z 417.345,A -85,B 0,C 180,E1 23565.057,E2 23565.057} C_VEL
LIN {X 0,Y 514.754,Z 420.088,A -85,B 0,C 180,E1 23564.509,E2 23564.509} C_VEL
LIN {X 0,Y 517.023,Z 422.711,A -85,B 0,C 180,E1 23563.484,E2 23563.484} C_VEL
LIN {X 0,Y 519.882,Z 424.243,A -85,B 0,C 180,E1 23562.367,E2 23562.367} C_VEL
LIN {X 0,Y 521.484,Z 427.47,A -85,B 0,C 180,E1 23561.672,E2 23561.672} C_VEL
LIN {X 0,Y 524.381,Z 429.983,A -85,B 0,C 180,E1 23560.623,E2 23560.623} C_VEL
LIN {X 0,Y 525.771,Z 430.862,A -85,B 0,C 180,E1 23560.156,E2 23560.156} C_VEL
LIN {X 0,Y 527.926,Z 434.393,A -85,B 0,C 180,E1 23559.373,E2 23559.373} C_VEL
LIN {X 0,Y 531.503,Z 437.48,A -85,B 0,C 180,E1 23558.247,E2 23558.247} C_VEL
LIN {X 0,Y 534.237,Z 441.358,A -85,B 0,C 180,E1 23557.38,E2 23557.38} C_VEL
LIN {X 0,Y 537.045,Z 443.901,A -85,B 0,C 180,E1 23556.578,E2 23556.578} C_VEL
LIN {X 0,Y 540.377,Z 448.152,A -85,B 0,C 180,E1 23555.63,E2 23555.63} C_VEL
LIN {X 0,Y 542.326,Z 450.099,A -85,B 0,C 180,E1 23555.113,E2 23555.113} C_VEL
LIN {X 0,Y 545.967,Z 454.571,A -85,B 0,C 180,E1 23554.159,E2 23554.159} C_VEL
LIN {X 0,Y 547.703,Z 456.596,A -85,B 0,C 180,E1 23553.723,E2 23553.723} C_VEL
LIN {X 0,Y 552.954,Z 462.928,A -85,B 0,C 180,E1 23552.454,E2 23552.454} C_VEL
LIN {X 0,Y 557.582,Z 468.669,A -85,B 0,C 180,E1 23551.393,E2 23551.393} C_VEL
LIN {X 0,Y 565.656,Z 478.758,A -85,B 0,C 180,E1 23549.661,E2 23549.661} C_VEL
LIN {X 0,Y 576.686,Z 493.285,A -85,B 0,C 180,E1 23547.487,E2 23547.487} C_VEL
LIN {X 0,Y 587.972,Z 508.997,A -85,B 0,C 180,E1 23545.449,E2 23545.449} C_VEL
LIN {X 0,Y 589.792,Z 511.797,A -85,B 0,C 180,E1 23545.131,E2 23545.131} C_VEL
LIN {X 0,Y 580.989,Z 726.771,A -85,B 0,C 180,E1 23541.934,E2 23541.934} C_VEL
LIN {X 0,Y 575.013,Z 876.888,A -85,B 0,C 180,E1 23539.717,E2 23539.717} C_VEL
LIN {X 0,Y 573.219,Z 901.562,A -85,B 0,C 180,E1 23539.251,E2 23539.251} C_VEL
LIN {X 0,Y 570.378,Z 929.434,A -85,B 0,C 180,E1 23538.534,E2 23538.534} C_VEL
LIN {X 0,Y 567.625,Z 951.407,A -85,B 0,C 180,E1 23537.82,E2 23537.82} C_VEL
LIN {X 0,Y 564.669,Z 972.028,A -85,B 0,C 180,E1 23537.02,E2 23537.02} C_VEL
LIN {X 0,Y 562.235,Z 987.347,A -85,B 0,C 180,E1 23536.34,E2 23536.34} C_VEL
LIN {X 0,Y 560.348,Z 994.496,A -85,B 0,C 180,E1 23536.074,E2 23536.074} C_VEL
LIN {X 0,Y 552.927,Z 1012.528,A -85,B 0,C 180,E1 23535.591,E2 23535.591} C_VEL
LIN {X 0,Y 550.88,Z 1019.321,A -85,B 0,C 180,E1 23535.269,E2 23535.269} C_VEL
LIN {X 0,Y 546.408,Z 1040.852,A -85,B 0,C 180,E1 23533.901,E2 23533.901} C_VEL
LIN {X 0,Y 542.343,Z 1059.295,A -85,B 0,C 180,E1 23532.57,E2 23532.57} C_VEL
LIN {X 0,Y 538.216,Z 1077.236,A -85,B 0,C 180,E1 23531.112,E2 23531.112} C_VEL
LIN {X 0,Y 533.498,Z 1097.194,A -85,B 0,C 180,E1 23529.281,E2 23529.281} C_VEL
LIN {X 0,Y 528.36,Z 1118.154,A -85,B 0,C 180,E1 23527.058,E2 23527.058} C_VEL
LIN {X 0,Y 524.431,Z 1134.044,A -85,B 0,C 180,E1 23525.147,E2 23525.147} C_VEL
LIN {X 0,Y 520.86,Z 1148.719,A -85,B 0,C 180,E1 23523.176,E2 23523.176} C_VEL
LIN {X 0,Y 517.132,Z 1164.43,A -85,B 0,C 180,E1 23520.815,E2 23520.815} C_VEL
LIN {X 0,Y 513.442,Z 1180.754,A -85,B 0,C 180,E1 23517.983,E2 23517.983} C_VEL
LIN {X 0,Y 510.542,Z 1194.836,A -85,B 0,C 180,E1 23515.2,E2 23515.2} C_VEL
LIN {X 0,Y 508.257,Z 1207.702,A -85,B 0,C 180,E1 23512.307,E2 23512.307} C_VEL
LIN {X 0,Y 506.58,Z 1218.35,A -85,B 0,C 180,E1 23509.479,E2 23509.479} C_VEL
LIN {X 0,Y 505.556,Z 1226.384,A -85,B 0,C 180,E1 23507.014,E2 23507.014} C_VEL
LIN {X 0,Y 504.845,Z 1232.943,A -85,B 0,C 180,E1 23504.679,E2 23504.679} C_VEL
LIN {X 0,Y 504.397,Z 1238.475,A -85,B 0,C 180,E1 23502.356,E2 23502.356} C_VEL
LIN {X 0,Y 504.1,Z 1243.239,A -85,B 0,C 180,E1 23499.931,E2 23499.931} C_VEL
LIN {X 0,Y 503.977,Z 1247.417,A -85,B 0,C 180,E1 23497.175,E2 23497.175} C_VEL
LIN {X 0,Y 503.917,Z 1250.445,A -85,B 0,C 180,E1 23494.091,E2 23494.091} C_VEL
LIN {X 0,Y 503.904,Z 1251.704,A -85,B 0,C 180,E1 23491.473,E2 23491.473} C_VEL
LIN {X 0,Y 503.869,Z 1251.834,A -85,B 0,C 180,E1 23489.085,E2 23489.085} C_VEL
LIN {X 0,Y 503.911,Z 1251.038,A -85,B 0,C 180,E1 23486.81,E2 23486.81} C_VEL
LIN {X 0,Y 503.931,Z 1249.237,A -85,B 0,C 180,E1 23484.416,E2 23484.416} C_VEL
LIN {X 0,Y 503.981,Z 1246.411,A -85,B 0,C 180,E1 23482.012,E2 23482.012} C_VEL
LIN {X 0,Y 504.176,Z 1242.348,A -85,B 0,C 180,E1 23479.483,E2 23479.483} C_VEL
LIN {X 0,Y 504.575,Z 1236.501,A -85,B 0,C 180,E1 23476.654,E2 23476.654} C_VEL
LIN {X 0,Y 505.373,Z 1228.036,A -85,B 0,C 180,E1 23473.442,E2 23473.442} C_VEL
LIN {X 0,Y 506.325,Z 1220.238,A -85,B 0,C 180,E1 23470.979,E2 23470.979} C_VEL
LIN {X 0,Y 507.605,Z 1211.666,A -85,B 0,C 180,E1 23468.624,E2 23468.624} C_VEL
LIN {X 0,Y 509.308,Z 1201.585,A -85,B 0,C 180,E1 23466.188,E2 23466.188} C_VEL
LIN {X 0,Y 511.94,Z 1187.991,A -85,B 0,C 180,E1 23463.302,E2 23463.302} C_VEL
LIN {X 0,Y 515.077,Z 1173.263,A -85,B 0,C 180,E1 23460.581,E2 23460.581} C_VEL
LIN {X 0,Y 518.08,Z 1160.345,A -85,B 0,C 180,E1 23458.461,E2 23458.461} C_VEL
LIN {X 0,Y 521.325,Z 1146.817,A -85,B 0,C 180,E1 23456.466,E2 23456.466} C_VEL
LIN {X 0,Y 525.354,Z 1130.383,A -85,B 0,C 180,E1 23454.297,E2 23454.297} C_VEL
LIN {X 0,Y 530.369,Z 1109.885,A -85,B 0,C 180,E1 23451.937,E2 23451.937} C_VEL
LIN {X 0,Y 534.632,Z 1092.307,A -85,B 0,C 180,E1 23450.163,E2 23450.163} C_VEL
LIN {X 0,Y 538.664,Z 1075.327,A -85,B 0,C 180,E1 23448.634,E2 23448.634} C_VEL
LIN {X 0,Y 542.948,Z 1056.644,A -85,B 0,C 180,E1 23447.135,E2 23447.135} C_VEL
LIN {X 0,Y 548.166,Z 1032.698,A -85,B 0,C 180,E1 23445.461,E2 23445.461} C_VEL
LIN {X 0,Y 552.497,Z 1010.701,A -85,B 0,C 180,E1 23444.15,E2 23444.15} C_VEL
LIN {X 0,Y 556.241,Z 990.114,A -85,B 0,C 180,E1 23443.085,E2 23443.085} C_VEL
LIN {X 0,Y 559.508,Z 970.357,A -85,B 0,C 180,E1 23442.202,E2 23442.202} C_VEL
LIN {X 0,Y 562.644,Z 948.979,A -85,B 0,C 180,E1 23441.383,E2 23441.383} C_VEL
LIN {X 0,Y 566.07,Z 921.457,A -85,B 0,C 180,E1 23440.528,E2 23440.528} C_VEL
LIN {X 0,Y 568.417,Z 896.918,A -85,B 0,C 180,E1 23439.942,E2 23439.942} C_VEL
LIN {X 0,Y 570.009,Z 874.978,A -85,B 0,C 180,E1 23439.542,E2 23439.542} C_VEL
LIN {X 0,Y 578.739,Z 663.705,A -85,B 0,C 180,E1 23436.405,E2 23436.405} C_VEL
LIN {X 0,Y 585.08,Z 515.93,A -85,B 0,C 180,E1 23434.185,E2 23434.185} C_VEL
LIN {X 0,Y 572.863,Z 498.771,A -85,B 0,C 180,E1 23431.929,E2 23431.929} C_VEL
LIN {X 0,Y 561.699,Z 483.983,A -85,B 0,C 180,E1 23429.662,E2 23429.662} C_VEL
LIN {X 0,Y 552.574,Z 472.544,A -85,B 0,C 180,E1 23427.625,E2 23427.625} C_VEL
LIN {X 0,Y 548.185,Z 467.188,A -85,B 0,C 180,E1 23426.573,E2 23426.573} C_VEL
LIN {X 0,Y 543.87,Z 461.889,A -85,B 0,C 180,E1 23425.481,E2 23425.481} C_VEL
LIN {X 0,Y 540.011,Z 457.052,A -85,B 0,C 180,E1 23424.446,E2 23424.446} C_VEL
LIN {X 0,Y 535.812,Z 452.466,A -85,B 0,C 180,E1 23423.276,E2 23423.276} C_VEL
LIN {X 0,Y 534.375,Z 450.577,A -85,B 0,C 180,E1 23422.846,E2 23422.846} C_VEL
LIN {X 0,Y 530.837,Z 446.945,A -85,B 0,C 180,E1 23421.782,E2 23421.782} C_VEL
LIN {X 0,Y 529.295,Z 444.534,A -85,B 0,C 180,E1 23421.267,E2 23421.267} C_VEL
LIN {X 0,Y 525.949,Z 441.619,A -85,B 0,C 180,E1 23420.185,E2 23420.185} C_VEL
LIN {X 0,Y 523.829,Z 438.214,A -85,B 0,C 180,E1 23419.398,E2 23419.398} C_VEL
LIN {X 0,Y 520.454,Z 435.71,A -85,B 0,C 180,E1 23418.192,E2 23418.192} C_VEL
LIN {X 0,Y 518.311,Z 432.143,A -85,B 0,C 180,E1 23417.283,E2 23417.283} C_VEL
LIN {X 0,Y 517.239,Z 431.399,A -85,B 0,C 180,E1 23416.856,E2 23416.856} C_VEL
LIN {X 0,Y 514.09,Z 428.921,A -85,B 0,C 180,E1 23415.512,E2 23415.512} C_VEL
LIN {X 0,Y 512.354,Z 425.732,A -85,B 0,C 180,E1 23414.61,E2 23414.61} C_VEL
LIN {X 0,Y 512.133,Z 424.991,A -85,B 0,C 180,E1 23414.472,E2 23414.472} C_VEL
LIN {X 0,Y 508.432,Z 423.146,A -85,B 0,C 180,E1 23412.609,E2 23412.609} C_VEL
LIN {X 0,Y 506.428,Z 420.322,A -85,B 0,C 180,E1 23411.33,E2 23411.33} C_VEL
LIN {X 0,Y 505.846,Z 418.184,A -85,B 0,C 180,E1 23410.824,E2 23410.824} C_VEL
LIN {X 0,Y 505.869,Z 418.167,A -85,B 0,C 180,E1 23407.267,E2 23407.267} C_VEL
LIN {X 0,Y 505.857,Z 418.153,A -85,B 0,C 180,E1 23403.74,E2 23403.74} C_VEL
LIN {X 0,Y 505.846,Z 418.206,A -85,B 0,C 180,E1 23400.227,E2 23400.227} C_VEL
LIN {X 0,Y 505.847,Z 418.145,A -85,B 0,C 180,E1 23396.714,E2 23396.714} C_VEL
LIN {X 0,Y 505.866,Z 418.203,A -85,B 0,C 180,E1 23393.189,E2 23393.189} C_VEL
LIN {X 0,Y 505.842,Z 418.157,A -85,B 0,C 180,E1 23389.752,E2 23389.752} C_VEL
LIN {X 0,Y 505.881,Z 418.379,A -85,B 0,C 180,E1 23389.552,E2 23389.552} C_VEL
LIN {X 0,Y 506.84,Z 421.137,A -85,B 0,C 180,E1 23388.795,E2 23388.795} C_VEL
LIN {X 0,Y 509.151,Z 423.728,A -85,B 0,C 180,E1 23387.409,E2 23387.409} C_VEL
LIN {X 0,Y 512.197,Z 425.201,A -85,B 0,C 180,E1 23385.905,E2 23385.905} C_VEL
LIN {X 0,Y 513.775,Z 428.502,A -85,B 0,C 180,E1 23385.056,E2 23385.056} C_VEL
LIN {X 0,Y 516.598,Z 431.059,A -85,B 0,C 180,E1 23383.816,E2 23383.816} C_VEL
LIN {X 0,Y 518.274,Z 432.101,A -85,B 0,C 180,E1 23383.15,E2 23383.15} C_VEL
LIN {X 0,Y 520.342,Z 435.623,A -85,B 0,C 180,E1 23382.267,E2 23382.267} C_VEL
LIN {X 0,Y 523.431,Z 438.395,A -85,B 0,C 180,E1 23381.137,E2 23381.137} C_VEL
LIN {X 0,Y 528.509,Z 444.663,A -85,B 0,C 180,E1 23379.368,E2 23379.368} C_VEL
LIN {X 0,Y 532.304,Z 449.035,A -85,B 0,C 180,E1 23378.165,E2 23378.165} C_VEL
LIN {X 0,Y 536.504,Z 454.491,A -85,B 0,C 180,E1 23376.901,E2 23376.901} C_VEL
LIN {X 0,Y 545.488,Z 466.044,A -85,B 0,C 180,E1 23374.455,E2 23374.455} C_VEL
LIN {X 0,Y 554.744,Z 478.543,A -85,B 0,C 180,E1 23372.2,E2 23372.2} C_VEL
LIN {X 0,Y 564.03,Z 491.48,A -85,B 0,C 180,E1 23370.152,E2 23370.152} C_VEL
LIN {X 0,Y 575.7,Z 508.698,A -85,B 0,C 180,E1 23367.807,E2 23367.807} C_VEL
LIN {X 0,Y 585.243,Z 523.812,A -85,B 0,C 180,E1 23366.039,E2 23366.039} C_VEL
LIN {X 0,Y 576.016,Z 742.488,A -85,B 0,C 180,E1 23362.771,E2 23362.771} C_VEL
LIN {X 0,Y 569.552,Z 900.925,A -85,B 0,C 180,E1 23360.42,E2 23360.42} C_VEL
LIN {X 0,Y 567.556,Z 926.796,A -85,B 0,C 180,E1 23359.938,E2 23359.938} C_VEL
LIN {X 0,Y 564.534,Z 954.462,A -85,B 0,C 180,E1 23359.234,E2 23359.234} C_VEL
LIN {X 0,Y 561.717,Z 976.027,A -85,B 0,C 180,E1 23358.542,E2 23358.542} C_VEL
LIN {X 0,Y 558.615,Z 996.838,A -85,B 0,C 180,E1 23357.747,E2 23357.747} C_VEL
LIN {X 0,Y 555.224,Z 1017.248,A -85,B 0,C 180,E1 23356.836,E2 23356.836} C_VEL
LIN {X 0,Y 550.694,Z 1042.317,A -85,B 0,C 180,E1 23355.529,E2 23355.529} C_VEL
LIN {X 0,Y 545.838,Z 1066.198,A -85,B 0,C 180,E1 23354.045,E2 23354.045} C_VEL
LIN {X 0,Y 541.635,Z 1085.811,A -85,B 0,C 180,E1 23352.652,E2 23352.652} C_VEL
LIN {X 0,Y 537.409,Z 1104.804,A -85,B 0,C 180,E1 23351.129,E2 23351.129} C_VEL
LIN {X 0,Y 532.413,Z 1126.802,A -85,B 0,C 180,E1 23349.129,E2 23349.129} C_VEL
LIN {X 0,Y 527.758,Z 1146.558,A -85,B 0,C 180,E1 23347.052,E2 23347.052} C_VEL
LIN {X 0,Y 524.044,Z 1162.395,A -85,B 0,C 180,E1 23345.189,E2 23345.189} C_VEL
LIN {X 0,Y 520.547,Z 1177.631,A -85,B 0,C 180,E1 23343.195,E2 23343.195} C_VEL
LIN {X 0,Y 516.781,Z 1194.552,A -85,B 0,C 180,E1 23340.721,E2 23340.721} C_VEL
LIN {X 0,Y 513.367,Z 1210.673,A -85,B 0,C 180,E1 23337.999,E2 23337.999} C_VEL
LIN {X 0,Y 511.118,Z 1221.81,A -85,B 0,C 180,E1 23335.869,E2 23335.869} C_VEL
LIN {X 0,Y 509.186,Z 1232.23,A -85,B 0,C 180,E1 23333.62,E2 23333.62} C_VEL
LIN {X 0,Y 507.562,Z 1241.955,A -85,B 0,C 180,E1 23331.257,E2 23331.257} C_VEL
LIN {X 0,Y 506.247,Z 1250.896,A -85,B 0,C 180,E1 23328.785,E2 23328.785} C_VEL
LIN {X 0,Y 505.119,Z 1260.609,A -85,B 0,C 180,E1 23325.622,E2 23325.622} C_VEL
LIN {X 0,Y 504.465,Z 1267.622,A -85,B 0,C 180,E1 23322.79,E2 23322.79} C_VEL
LIN {X 0,Y 504.15,Z 1272.681,A -85,B 0,C 180,E1 23320.287,E2 23320.287} C_VEL
LIN {X 0,Y 503.969,Z 1276.667,A -85,B 0,C 180,E1 23317.758,E2 23317.758} C_VEL
LIN {X 0,Y 503.925,Z 1279.533,A -85,B 0,C 180,E1 23315.242,E2 23315.242} C_VEL
LIN {X 0,Y 503.909,Z 1281.575,A -85,B 0,C 180,E1 23312.166,E2 23312.166} C_VEL
LIN {X 0,Y 503.865,Z 1281.872,A -85,B 0,C 180,E1 23309.323,E2 23309.323} C_VEL
LIN {X 0,Y 503.91,Z 1281.085,A -85,B 0,C 180,E1 23306.934,E2 23306.934} C_VEL
LIN {X 0,Y 503.929,Z 1279.315,A -85,B 0,C 180,E1 23304.54,E2 23304.54} C_VEL
LIN {X 0,Y 503.973,Z 1276.521,A -85,B 0,C 180,E1 23302.137,E2 23302.137} C_VEL
LIN {X 0,Y 504.166,Z 1272.493,A -85,B 0,C 180,E1 23299.608,E2 23299.608} C_VEL
LIN {X 0,Y 504.495,Z 1267.302,A -85,B 0,C 180,E1 23297.064,E2 23297.064} C_VEL
LIN {X 0,Y 505.206,Z 1259.697,A -85,B 0,C 180,E1 23294.038,E2 23294.038} C_VEL
LIN {X 0,Y 506.301,Z 1250.433,A -85,B 0,C 180,E1 23291.081,E2 23291.081} C_VEL
LIN {X 0,Y 507.583,Z 1241.838,A -85,B 0,C 180,E1 23288.712,E2 23288.712} C_VEL
LIN {X 0,Y 509.275,Z 1231.769,A -85,B 0,C 180,E1 23286.273,E2 23286.273} C_VEL
LIN {X 0,Y 511.849,Z 1218.428,A -85,B 0,C 180,E1 23283.434,E2 23283.434} C_VEL
LIN {X 0,Y 514.915,Z 1203.085,A -85,B 0,C 180,E1 23280.68,E2 23280.68} C_VEL
LIN {X 0,Y 517.782,Z 1189.921,A -85,B 0,C 180,E1 23278.582,E2 23278.582} C_VEL
LIN {X 0,Y 520.923,Z 1175.992,A -85,B 0,C 180,E1 23276.581,E2 23276.581} C_VEL
LIN {X 0,Y 524.578,Z 1160.133,A -85,B 0,C 180,E1 23274.53,E2 23274.53} C_VEL
LIN {X 0,Y 529.516,Z 1139.035,A -85,B 0,C 180,E1 23272.122,E2 23272.122} C_VEL
LIN {X 0,Y 534.026,Z 1119.577,A -85,B 0,C 180,E1 23270.192,E2 23270.192} C_VEL
LIN {X 0,Y 538.144,Z 1101.542,A -85,B 0,C 180,E1 23268.598,E2 23268.598} C_VEL
LIN {X 0,Y 542.434,Z 1082.223,A -85,B 0,C 180,E1 23267.079,E2 23267.079} C_VEL
LIN {X 0,Y 547.768,Z 1057.023,A -85,B 0,C 180,E1 23265.36,E2 23265.36} C_VEL
LIN {X 0,Y 551.951,Z 1035.412,A -85,B 0,C 180,E1 23264.097,E2 23264.097} C_VEL
LIN {X 0,Y 555.574,Z 1015.16,A -85,B 0,C 180,E1 23263.066,E2 23263.066} C_VEL
LIN {X 0,Y 558.977,Z 994.455,A -85,B 0,C 180,E1 23262.156,E2 23262.156} C_VEL
LIN {X 0,Y 562.433,Z 970.974,A -85,B 0,C 180,E1 23261.281,E2 23261.281} C_VEL
LIN {X 0,Y 565.887,Z 942.661,A -85,B 0,C 180,E1 23260.444,E2 23260.444} C_VEL
LIN {X 0,Y 568.098,Z 920.172,A -85,B 0,C 180,E1 23259.931,E2 23259.931} C_VEL
LIN {X 0,Y 569.708,Z 897.866,A -85,B 0,C 180,E1 23259.533,E2 23259.533} C_VEL
LIN {X 0,Y 578.529,Z 680.561,A -85,B 0,C 180,E1 23256.311,E2 23256.311} C_VEL
LIN {X 0,Y 585.168,Z 523.663,A -85,B 0,C 180,E1 23253.955,E2 23253.955} C_VEL
LIN {X 0,Y 575.188,Z 508.005,A -85,B 0,C 180,E1 23252.108,E2 23252.108} C_VEL
LIN {X 0,Y 563.318,Z 490.504,A -85,B 0,C 180,E1 23249.714,E2 23249.714} C_VEL
LIN {X 0,Y 552.644,Z 475.655,A -85,B 0,C 180,E1 23247.33,E2 23247.33} C_VEL
LIN {X 0,Y 543.598,Z 463.729,A -85,B 0,C 180,E1 23245.086,E2 23245.086} C_VEL
LIN {X 0,Y 536.217,Z 454.247,A -85,B 0,C 180,E1 23243.054,E2 23243.054} C_VEL
LIN {X 0,Y 531.673,Z 448.533,A -85,B 0,C 180,E1 23241.688,E2 23241.688} C_VEL
LIN {X 0,Y 528.014,Z 443.927,A -85,B 0,C 180,E1 23240.508,E2 23240.508} C_VEL
LIN {X 0,Y 522.638,Z 437.635,A -85,B 0,C 180,E1 23238.633,E2 23238.633} C_VEL
LIN {X 0,Y 519.666,Z 434.809,A -85,B 0,C 180,E1 23237.525,E2 23237.525} C_VEL
LIN {X 0,Y 517.797,Z 431.651,A -85,B 0,C 180,E1 23236.722,E2 23236.722} C_VEL
LIN {X 0,Y 514.546,Z 429.466,A -85,B 0,C 180,E1 23235.382,E2 23235.382} C_VEL
LIN {X 0,Y 512.502,Z 426.339,A -85,B 0,C 180,E1 23234.375,E2 23234.375} C_VEL
LIN {X 0,Y 511.976,Z 424.986,A -85,B 0,C 180,E1 23234.073,E2 23234.073} C_VEL
LIN {X 0,Y 508.362,Z 423.182,A -85,B 0,C 180,E1 23232.264,E2 23232.264} C_VEL
LIN {X 0,Y 506.271,Z 420.081,A -85,B 0,C 180,E1 23230.93,E2 23230.93} C_VEL
LIN {X 0,Y 505.767,Z 418.177,A -85,B 0,C 180,E1 23230.479,E2 23230.479} C_VEL
LIN {X 0,Y 505.829,Z 418.187,A -85,B 0,C 180,E1 23227.154,E2 23227.154} C_VEL
LIN {X 0,Y 505.772,Z 418.162,A -85,B 0,C 180,E1 23223.854,E2 23223.854} C_VEL
LIN {X 0,Y 505.784,Z 418.225,A -85,B 0,C 180,E1 23220.34,E2 23220.34} C_VEL
LIN {X 0,Y 505.834,Z 418.148,A -85,B 0,C 180,E1 23217.054,E2 23217.054} C_VEL
LIN {X 0,Y 505.795,Z 418.223,A -85,B 0,C 180,E1 23213.644,E2 23213.644} C_VEL
LIN {X 0,Y 505.796,Z 418.16,A -85,B 0,C 180,E1 23210.097,E2 23210.097} C_VEL
LIN {X 0,Y 505.875,Z 418.389,A -85,B 0,C 180,E1 23208.918,E2 23208.918} C_VEL
LIN {X 0,Y 506.841,Z 421.263,A -85,B 0,C 180,E1 23208.16,E2 23208.16} C_VEL
LIN {X 0,Y 509.099,Z 423.669,A -85,B 0,C 180,E1 23206.831,E2 23206.831} C_VEL
LIN {X 0,Y 512.215,Z 425.304,A -85,B 0,C 180,E1 23205.299,E2 23205.299} C_VEL
LIN {X 0,Y 513.868,Z 428.695,A -85,B 0,C 180,E1 23204.424,E2 23204.424} C_VEL
LIN {X 0,Y 516.602,Z 431.088,A -85,B 0,C 180,E1 23203.238,E2 23203.238} C_VEL
LIN {X 0,Y 518.223,Z 432.076,A -85,B 0,C 180,E1 23202.598,E2 23202.598} C_VEL
LIN {X 0,Y 520.235,Z 435.523,A -85,B 0,C 180,E1 23201.743,E2 23201.743} C_VEL
LIN {X 0,Y 523.76,Z 438.187,A -85,B 0,C 180,E1 23200.483,E2 23200.483} C_VEL
LIN {X 0,Y 526.654,Z 442.443,A -85,B 0,C 180,E1 23199.437,E2 23199.437} C_VEL
LIN {X 0,Y 529.635,Z 445.07,A -85,B 0,C 180,E1 23198.486,E2 23198.486} C_VEL
LIN {X 0,Y 532.604,Z 449.073,A -85,B 0,C 180,E1 23197.54,E2 23197.54} C_VEL
LIN {X 0,Y 535.033,Z 451.338,A -85,B 0,C 180,E1 23196.834,E2 23196.834} C_VEL
LIN {X 0,Y 538.515,Z 455.697,A -85,B 0,C 180,E1 23195.832,E2 23195.832} C_VEL
LIN {X 0,Y 540.341,Z 457.674,A -85,B 0,C 180,E1 23195.337,E2 23195.337} C_VEL
LIN {X 0,Y 544.252,Z 462.295,A -85,B 0,C 180,E1 23194.305,E2 23194.305} C_VEL
LIN {X 0,Y 549.3,Z 468.334,A -85,B 0,C 180,E1 23193.047,E2 23193.047} C_VEL
LIN {X 0,Y 559.045,Z 480.704,A -85,B 0,C 180,E1 23190.802,E2 23190.802} C_VEL
LIN {X 0,Y 570.065,Z 494.982,A -85,B 0,C 180,E1 23188.516,E2 23188.516} C_VEL
LIN {X 0,Y 583.211,Z 513.218,A -85,B 0,C 180,E1 23186.049,E2 23186.049} C_VEL
LIN {X 0,Y 585.065,Z 516.215,A -85,B 0,C 180,E1 23185.713,E2 23185.713} C_VEL
LIN {X 0,Y 575.925,Z 731.045,A -85,B 0,C 180,E1 23182.502,E2 23182.502} C_VEL
LIN {X 0,Y 569.868,Z 877.208,A -85,B 0,C 180,E1 23180.33,E2 23180.33} C_VEL
LIN {X 0,Y 567.994,Z 902.169,A -85,B 0,C 180,E1 23179.857,E2 23179.857} C_VEL
LIN {X 0,Y 565.074,Z 929.819,A -85,B 0,C 180,E1 23179.142,E2 23179.142} C_VEL
LIN {X 0,Y 562.341,Z 951,A -85,B 0,C 180,E1 23178.453,E2 23178.453} C_VEL
LIN {X 0,Y 559.302,Z 971.595,A -85,B 0,C 180,E1 23177.655,E2 23177.655} C_VEL
LIN {X 0,Y 555.95,Z 991.796,A -85,B 0,C 180,E1 23176.742,E2 23176.742} C_VEL
LIN {X 0,Y 551.793,Z 1014.545,A -85,B 0,C 180,E1 23175.548,E2 23175.548} C_VEL
LIN {X 0,Y 550.88,Z 1019.321,A -85,B 0,C 180,E1 23175.269,E2 23175.269} C_VEL
LIN {X 0,Y 548.776,Z 1026.205,A -85,B 0,C 180,E1 23174.928,E2 23174.928} C_VEL
LIN {X 0,Y 540.754,Z 1043.534,A -85,B 0,C 180,E1 23174.263,E2 23174.263} C_VEL
LIN {X 0,Y 538.617,Z 1049.933,A -85,B 0,C 180,E1 23173.89,E2 23173.89} C_VEL
LIN {X 0,Y 533.172,Z 1072.894,A -85,B 0,C 180,E1 23172.091,E2 23172.091} C_VEL
LIN {X 0,Y 528.893,Z 1090.296,A -85,B 0,C 180,E1 23170.536,E2 23170.536} C_VEL
LIN {X 0,Y 524.717,Z 1106.806,A -85,B 0,C 180,E1 23168.885,E2 23168.885} C_VEL
LIN {X 0,Y 520.581,Z 1122.927,A -85,B 0,C 180,E1 23167.084,E2 23167.084} C_VEL
LIN {X 0,Y 515.796,Z 1141.714,A -85,B 0,C 180,E1 23164.72,E2 23164.72} C_VEL
LIN {X 0,Y 511.456,Z 1158.654,A -85,B 0,C 180,E1 23162.248,E2 23162.248} C_VEL
LIN {X 0,Y 508.169,Z 1172.154,A -85,B 0,C 180,E1 23160.03,E2 23160.03} C_VEL
LIN {X 0,Y 505.357,Z 1184.194,A -85,B 0,C 180,E1 23157.818,E2 23157.818} C_VEL
LIN {X 0,Y 502.526,Z 1197.472,A -85,B 0,C 180,E1 23155.068,E2 23155.068} C_VEL
LIN {X 0,Y 500.063,Z 1210.456,A -85,B 0,C 180,E1 23151.95,E2 23151.95} C_VEL
LIN {X 0,Y 498.637,Z 1219.258,A -85,B 0,C 180,E1 23149.529,E2 23149.529} C_VEL
LIN {X 0,Y 497.632,Z 1226.739,A -85,B 0,C 180,E1 23147.173,E2 23147.173} C_VEL
LIN {X 0,Y 496.858,Z 1233.55,A -85,B 0,C 180,E1 23144.682,E2 23144.682} C_VEL
LIN {X 0,Y 496.347,Z 1240.002,A -85,B 0,C 180,E1 23141.851,E2 23141.851} C_VEL
LIN {X 0,Y 496.041,Z 1245.658,A -85,B 0,C 180,E1 23138.573,E2 23138.573} C_VEL
LIN {X 0,Y 495.946,Z 1248.813,A -85,B 0,C 180,E1 23136.012,E2 23136.012} C_VEL
LIN {X 0,Y 495.913,Z 1250.788,A -85,B 0,C 180,E1 23133.575,E2 23133.575} C_VEL
LIN {X 0,Y 495.896,Z 1251.75,A -85,B 0,C 180,E1 23131.266,E2 23131.266} C_VEL
LIN {X 0,Y 495.875,Z 1251.811,A -85,B 0,C 180,E1 23128.955,E2 23128.955} C_VEL
LIN {X 0,Y 495.912,Z 1250.969,A -85,B 0,C 180,E1 23126.643,E2 23126.643} C_VEL
LIN {X 0,Y 495.938,Z 1249.12,A -85,B 0,C 180,E1 23124.209,E2 23124.209} C_VEL
LIN {X 0,Y 496,Z 1246.247,A -85,B 0,C 180,E1 23121.766,E2 23121.766} C_VEL
LIN {X 0,Y 496.216,Z 1241.931,A -85,B 0,C 180,E1 23119.077,E2 23119.077} C_VEL
LIN {X 0,Y 496.705,Z 1235.267,A -85,B 0,C 180,E1 23115.898,E2 23115.898} C_VEL
LIN {X 0,Y 497.57,Z 1227.326,A -85,B 0,C 180,E1 23112.934,E2 23112.934} C_VEL
LIN {X 0,Y 498.581,Z 1219.625,A -85,B 0,C 180,E1 23110.489,E2 23110.489} C_VEL
LIN {X 0,Y 499.959,Z 1211.071,A -85,B 0,C 180,E1 23108.122,E2 23108.122} C_VEL
LIN {X 0,Y 502.021,Z 1199.864,A -85,B 0,C 180,E1 23105.396,E2 23105.396} C_VEL
LIN {X 0,Y 505.002,Z 1185.767,A -85,B 0,C 180,E1 23102.395,E2 23102.395} C_VEL
LIN {X 0,Y 507.999,Z 1172.844,A -85,B 0,C 180,E1 23100,E2 23100} C_VEL
LIN {X 0,Y 511.16,Z 1159.858,A -85,B 0,C 180,E1 23097.851,E2 23097.851} C_VEL
LIN {X 0,Y 514.811,Z 1145.422,A -85,B 0,C 180,E1 23095.715,E2 23095.715} C_VEL
LIN {X 0,Y 519.935,Z 1125.486,A -85,B 0,C 180,E1 23093.126,E2 23093.126} C_VEL
LIN {X 0,Y 524.419,Z 1107.959,A -85,B 0,C 180,E1 23091.146,E2 23091.146} C_VEL
LIN {X 0,Y 528.52,Z 1091.754,A -85,B 0,C 180,E1 23089.511,E2 23089.511} C_VEL
LIN {X 0,Y 532.833,Z 1074.271,A -85,B 0,C 180,E1 23087.935,E2 23087.935} C_VEL
LIN {X 0,Y 538.083,Z 1052.354,A -85,B 0,C 180,E1 23086.192,E2 23086.192} C_VEL
LIN {X 0,Y 543.11,Z 1029.387,A -85,B 0,C 180,E1 23084.634,E2 23084.634} C_VEL
LIN {X 0,Y 547.076,Z 1009.864,A -85,B 0,C 180,E1 23083.478,E2 23083.478} C_VEL
LIN {X 0,Y 550.822,Z 989.849,A -85,B 0,C 180,E1 23082.443,E2 23082.443} C_VEL
LIN {X 0,Y 554.317,Z 969.334,A -85,B 0,C 180,E1 23081.529,E2 23081.529} C_VEL
LIN {X 0,Y 558.158,Z 943.863,A -85,B 0,C 180,E1 23080.572,E2 23080.572} C_VEL
LIN {X 0,Y 561.288,Z 917.771,A -85,B 0,C 180,E1 23079.802,E2 23079.802} C_VEL
LIN {X 0,Y 563.407,Z 895.954,A -85,B 0,C 180,E1 23079.292,E2 23079.292} C_VEL
LIN {X 0,Y 565.012,Z 874.039,A -85,B 0,C 180,E1 23078.897,E2 23078.897} C_VEL
LIN {X 0,Y 574.297,Z 657.583,A -85,B 0,C 180,E1 23075.666,E2 23075.666} C_VEL
LIN {X 0,Y 580.417,Z 520.284,A -85,B 0,C 180,E1 23073.592,E2 23073.592} C_VEL
LIN {X 0,Y 568.794,Z 504.006,A -85,B 0,C 180,E1 23071.385,E2 23071.385} C_VEL
LIN {X 0,Y 559.005,Z 490.878,A -85,B 0,C 180,E1 23069.347,E2 23069.347} C_VEL
LIN {X 0,Y 550.091,Z 479.572,A -85,B 0,C 180,E1 23067.32,E2 23067.32} C_VEL
LIN {X 0,Y 545.656,Z 474.126,A -85,B 0,C 180,E1 23066.237,E2 23066.237} C_VEL
LIN {X 0,Y 541.587,Z 469.068,A -85,B 0,C 180,E1 23065.186,E2 23065.186} C_VEL
LIN {X 0,Y 537.045,Z 463.577,A -85,B 0,C 180,E1 23063.946,E2 23063.946} C_VEL
LIN {X 0,Y 533.233,Z 458.974,A -85,B 0,C 180,E1 23062.84,E2 23062.84} C_VEL
LIN {X 0,Y 528.589,Z 453.857,A -85,B 0,C 180,E1 23061.413,E2 23061.413} C_VEL
LIN {X 0,Y 527.2,Z 451.923,A -85,B 0,C 180,E1 23060.948,E2 23060.948} C_VEL
LIN {X 0,Y 523.718,Z 448.496,A -85,B 0,C 180,E1 23059.78,E2 23059.78} C_VEL
LIN {X 0,Y 521.971,Z 445.794,A -85,B 0,C 180,E1 23059.121,E2 23059.121} C_VEL
LIN {X 0,Y 518.673,Z 443.095,A -85,B 0,C 180,E1 23057.908,E2 23057.908} C_VEL
LIN {X 0,Y 516.299,Z 439.4,A -85,B 0,C 180,E1 23056.888,E2 23056.888} C_VEL
LIN {X 0,Y 512.884,Z 436.888,A -85,B 0,C 180,E1 23055.433,E2 23055.433} C_VEL
LIN {X 0,Y 510.827,Z 433.393,A -85,B 0,C 180,E1 23054.365,E2 23054.365} C_VEL
LIN {X 0,Y 510.477,Z 432.761,A -85,B 0,C 180,E1 23054.173,E2 23054.173} C_VEL
LIN {X 0,Y 506.894,Z 430.672,A -85,B 0,C 180,E1 23052.301,E2 23052.301} C_VEL
LIN {X 0,Y 504.969,Z 427.69,A -85,B 0,C 180,E1 23051.016,E2 23051.016} C_VEL
LIN {X 0,Y 504.345,Z 426.03,A -85,B 0,C 180,E1 23050.509,E2 23050.509} C_VEL
LIN {X 0,Y 500.35,Z 423.959,A -85,B 0,C 180,E1 23047.348,E2 23047.348} C_VEL
LIN {X 0,Y 498.155,Z 420.372,A -85,B 0,C 180,E1 23044.259,E2 23044.259} C_VEL
LIN {X 0,Y 497.917,Z 419.135,A -85,B 0,C 180,E1 23043.454,E2 23043.454} C_VEL
LIN {X 0,Y 497.928,Z 419.206,A -85,B 0,C 180,E1 23039.885,E2 23039.885} C_VEL
LIN {X 0,Y 497.935,Z 419.308,A -85,B 0,C 180,E1 23036.777,E2 23036.777} C_VEL
LIN {X 0,Y 499.581,Z 423.185,A -85,B 0,C 180,E1 23033.911,E2 23033.911} C_VEL
LIN {X 0,Y 503.28,Z 425.721,A -85,B 0,C 180,E1 23030.624,E2 23030.624} C_VEL
LIN {X 0,Y 504.521,Z 426.23,A -85,B 0,C 180,E1 23029.783,E2 23029.783} C_VEL
LIN {X 0,Y 505.848,Z 429.378,A -85,B 0,C 180,E1 23028.773,E2 23028.773} C_VEL
LIN {X 0,Y 508.398,Z 431.869,A -85,B 0,C 180,E1 23027.275,E2 23027.275} C_VEL
LIN {X 0,Y 510.711,Z 433.04,A -85,B 0,C 180,E1 23026.123,E2 23026.123} C_VEL
LIN {X 0,Y 512.566,Z 436.492,A -85,B 0,C 180,E1 23025.136,E2 23025.136} C_VEL
LIN {X 0,Y 515.652,Z 439.08,A -85,B 0,C 180,E1 23023.786,E2 23023.786} C_VEL
LIN {X 0,Y 516.701,Z 439.898,A -85,B 0,C 180,E1 23023.357,E2 23023.357} C_VEL
LIN {X 0,Y 519.099,Z 443.62,A -85,B 0,C 180,E1 23022.339,E2 23022.339} C_VEL
LIN {X 0,Y 521.876,Z 446.179,A -85,B 0,C 180,E1 23021.31,E2 23021.31} C_VEL
LIN {X 0,Y 526.601,Z 452.035,A -85,B 0,C 180,E1 23019.638,E2 23019.638} C_VEL
LIN {X 0,Y 531.134,Z 457.659,A -85,B 0,C 180,E1 23018.173,E2 23018.173} C_VEL
LIN {X 0,Y 536.124,Z 464.021,A -85,B 0,C 180,E1 23016.681,E2 23016.681} C_VEL
LIN {X 0,Y 543.735,Z 474.043,A -85,B 0,C 180,E1 23014.6,E2 23014.6} C_VEL
LIN {X 0,Y 551.717,Z 484.824,A -85,B 0,C 180,E1 23012.624,E2 23012.624} C_VEL
LIN {X 0,Y 561.194,Z 498.209,A -85,B 0,C 180,E1 23010.485,E2 23010.485} C_VEL
LIN {X 0,Y 572.616,Z 515.272,A -85,B 0,C 180,E1 23008.144,E2 23008.144} C_VEL
LIN {X 0,Y 580.571,Z 528.006,A -85,B 0,C 180,E1 23006.632,E2 23006.632} C_VEL
LIN {X 0,Y 571.064,Z 744.924,A -85,B 0,C 180,E1 23003.375,E2 23003.375} C_VEL
LIN {X 0,Y 564.456,Z 900.677,A -85,B 0,C 180,E1 23001.049,E2 23001.049} C_VEL
LIN {X 0,Y 562.384,Z 926.707,A -85,B 0,C 180,E1 23000.564,E2 23000.564} C_VEL
LIN {X 0,Y 559.264,Z 954.314,A -85,B 0,C 180,E1 22999.859,E2 22999.859} C_VEL
LIN {X 0,Y 556.367,Z 975.767,A -85,B 0,C 180,E1 22999.17,E2 22999.17} C_VEL
LIN {X 0,Y 553.153,Z 996.576,A -85,B 0,C 180,E1 22998.373,E2 22998.373} C_VEL
LIN {X 0,Y 549.642,Z 1016.984,A -85,B 0,C 180,E1 22997.46,E2 22997.46} C_VEL
LIN {X 0,Y 544.943,Z 1042.051,A -85,B 0,C 180,E1 22996.148,E2 22996.148} C_VEL
LIN {X 0,Y 539.958,Z 1065.661,A -85,B 0,C 180,E1 22994.676,E2 22994.676} C_VEL
LIN {X 0,Y 535.58,Z 1085.335,A -85,B 0,C 180,E1 22993.272,E2 22993.272} C_VEL
LIN {X 0,Y 531.291,Z 1103.855,A -85,B 0,C 180,E1 22991.78,E2 22991.78} C_VEL
LIN {X 0,Y 526.189,Z 1125.35,A -85,B 0,C 180,E1 22989.824,E2 22989.824} C_VEL
LIN {X 0,Y 521.155,Z 1145.84,A -85,B 0,C 180,E1 22987.661,E2 22987.661} C_VEL
LIN {X 0,Y 517.156,Z 1162.118,A -85,B 0,C 180,E1 22985.729,E2 22985.729} C_VEL
LIN {X 0,Y 513.493,Z 1177.353,A -85,B 0,C 180,E1 22983.712,E2 22983.712} C_VEL
LIN {X 0,Y 509.47,Z 1194.561,A -85,B 0,C 180,E1 22981.163,E2 22981.163} C_VEL
LIN {X 0,Y 505.894,Z 1210.582,A -85,B 0,C 180,E1 22978.413,E2 22978.413} C_VEL
LIN {X 0,Y 503.335,Z 1222.81,A -85,B 0,C 180,E1 22976.046,E2 22976.046} C_VEL
LIN {X 0,Y 501.55,Z 1232.228,A -85,B 0,C 180,E1 22974.002,E2 22974.002} C_VEL
LIN {X 0,Y 499.814,Z 1241.953,A -85,B 0,C 180,E1 22971.603,E2 22971.603} C_VEL
LIN {X 0,Y 498.409,Z 1250.894,A -85,B 0,C 180,E1 22969.091,E2 22969.091} C_VEL
LIN {X 0,Y 497.233,Z 1260.304,A -85,B 0,C 180,E1 22965.996,E2 22965.996} C_VEL
LIN {X 0,Y 496.525,Z 1267.533,A -85,B 0,C 180,E1 22963.039,E2 22963.039} C_VEL
LIN {X 0,Y 496.192,Z 1272.471,A -85,B 0,C 180,E1 22960.571,E2 22960.571} C_VEL
LIN {X 0,Y 495.984,Z 1276.505,A -85,B 0,C 180,E1 22958.001,E2 22958.001} C_VEL
LIN {X 0,Y 495.93,Z 1279.303,A -85,B 0,C 180,E1 22955.559,E2 22955.559} C_VEL
LIN {X 0,Y 495.91,Z 1281.147,A -85,B 0,C 180,E1 22953.01,E2 22953.01} C_VEL
LIN {X 0,Y 495.903,Z 1282,A -85,B 0,C 180,E1 22950.005,E2 22950.005} C_VEL
LIN {X 0,Y 495.909,Z 1281.153,A -85,B 0,C 180,E1 22947,E2 22947} C_VEL
LIN {X 0,Y 495.932,Z 1279.312,A -85,B 0,C 180,E1 22944.452,E2 22944.452} C_VEL
LIN {X 0,Y 495.981,Z 1276.518,A -85,B 0,C 180,E1 22942.01,E2 22942.01} C_VEL
LIN {X 0,Y 496.191,Z 1272.49,A -85,B 0,C 180,E1 22939.439,E2 22939.439} C_VEL
LIN {X 0,Y 496.548,Z 1267.302,A -85,B 0,C 180,E1 22936.854,E2 22936.854} C_VEL
LIN {X 0,Y 497.337,Z 1259.343,A -85,B 0,C 180,E1 22933.659,E2 22933.659} C_VEL
LIN {X 0,Y 498.456,Z 1250.525,A -85,B 0,C 180,E1 22930.8,E2 22930.8} C_VEL
LIN {X 0,Y 499.807,Z 1241.999,A -85,B 0,C 180,E1 22928.408,E2 22928.408} C_VEL
LIN {X 0,Y 501.543,Z 1232.282,A -85,B 0,C 180,E1 22926.01,E2 22926.01} C_VEL
LIN {X 0,Y 503.428,Z 1222.375,A -85,B 0,C 180,E1 22923.864,E2 22923.864} C_VEL
LIN {X 0,Y 506.058,Z 1209.811,A -85,B 0,C 180,E1 22921.443,E2 22921.443} C_VEL
LIN {X 0,Y 510.048,Z 1191.995,A -85,B 0,C 180,E1 22918.446,E2 22918.446} C_VEL
LIN {X 0,Y 513.584,Z 1176.971,A -85,B 0,C 180,E1 22916.235,E2 22916.235} C_VEL
LIN {X 0,Y 517.252,Z 1161.735,A -85,B 0,C 180,E1 22914.223,E2 22914.223} C_VEL
LIN {X 0,Y 521.276,Z 1145.349,A -85,B 0,C 180,E1 22912.282,E2 22912.282} C_VEL
LIN {X 0,Y 526.584,Z 1123.613,A -85,B 0,C 180,E1 22910.012,E2 22910.012} C_VEL
LIN {X 0,Y 531.259,Z 1103.968,A -85,B 0,C 180,E1 22908.23,E2 22908.23} C_VEL
LIN {X 0,Y 535.575,Z 1085.329,A -85,B 0,C 180,E1 22906.728,E2 22906.728} C_VEL
LIN {X 0,Y 540.046,Z 1065.242,A -85,B 0,C 180,E1 22905.296,E2 22905.296} C_VEL
LIN {X 0,Y 545.374,Z 1039.724,A -85,B 0,C 180,E1 22903.725,E2 22903.725} C_VEL
LIN {X 0,Y 549.6,Z 1017.163,A -85,B 0,C 180,E1 22902.55,E2 22902.55} C_VEL
LIN {X 0,Y 553.107,Z 996.767,A -85,B 0,C 180,E1 22901.636,E2 22901.636} C_VEL
LIN {X 0,Y 556.319,Z 975.981,A -85,B 0,C 180,E1 22900.839,E2 22900.839} C_VEL
LIN {X 0,Y 559.304,Z 953.908,A -85,B 0,C 180,E1 22900.13,E2 22900.13} C_VEL
LIN {X 0,Y 562.454,Z 925.694,A -85,B 0,C 180,E1 22899.417,E2 22899.417} C_VEL
LIN {X 0,Y 564.448,Z 900.485,A -85,B 0,C 180,E1 22898.949,E2 22898.949} C_VEL
LIN {X 0,Y 572.342,Z 714.235,A -85,B 0,C 180,E1 22896.17,E2 22896.17} C_VEL
LIN {X 0,Y 580.487,Z 527.849,A -85,B 0,C 180,E1 22893.361,E2 22893.361} C_VEL
LIN {X 0,Y 571.417,Z 513.568,A -85,B 0,C 180,E1 22891.636,E2 22891.636} C_VEL
LIN {X 0,Y 560.595,Z 497.379,A -85,B 0,C 180,E1 22889.403,E2 22889.403} C_VEL
LIN {X 0,Y 549.948,Z 482.432,A -85,B 0,C 180,E1 22886.977,E2 22886.977} C_VEL
LIN {X 0,Y 541.127,Z 470.642,A -85,B 0,C 180,E1 22884.742,E2 22884.742} C_VEL
LIN {X 0,Y 534.204,Z 461.611,A -85,B 0,C 180,E1 22882.796,E2 22882.796} C_VEL
LIN {X 0,Y 529.55,Z 455.752,A -85,B 0,C 180,E1 22881.372,E2 22881.372} C_VEL
LIN {X 0,Y 525.025,Z 450.166,A -85,B 0,C 180,E1 22879.874,E2 22879.874} C_VEL
LIN {X 0,Y 521.097,Z 445.339,A -85,B 0,C 180,E1 22878.458,E2 22878.458} C_VEL
LIN {X 0,Y 518.023,Z 442.356,A -85,B 0,C 180,E1 22877.293,E2 22877.293} C_VEL
LIN {X 0,Y 516.302,Z 439.421,A -85,B 0,C 180,E1 22876.54,E2 22876.54} C_VEL
LIN {X 0,Y 512.982,Z 437.022,A -85,B 0,C 180,E1 22875.141,E2 22875.141} C_VEL
LIN {X 0,Y 510.875,Z 433.714,A -85,B 0,C 180,E1 22874.075,E2 22874.075} C_VEL
LIN {X 0,Y 510.433,Z 432.785,A -85,B 0,C 180,E1 22873.827,E2 22873.827} C_VEL
LIN {X 0,Y 506.817,Z 430.704,A -85,B 0,C 180,E1 22871.956,E2 22871.956} C_VEL
LIN {X 0,Y 504.738,Z 427.253,A -85,B 0,C 180,E1 22870.559,E2 22870.559} C_VEL
LIN {X 0,Y 504.242,Z 426.022,A -85,B 0,C 180,E1 22870.165,E2 22870.165} C_VEL
LIN {X 0,Y 500.431,Z 424.081,A -85,B 0,C 180,E1 22867.231,E2 22867.231} C_VEL
LIN {X 0,Y 498.261,Z 420.924,A -85,B 0,C 180,E1 22864.489,E2 22864.489} C_VEL
LIN {X 0,Y 497.862,Z 419.14,A -85,B 0,C 180,E1 22863.454,E2 22863.454} C_VEL
LIN {X 0,Y 497.842,Z 419.22,A -85,B 0,C 180,E1 22860.115,E2 22860.115} C_VEL
LIN {X 0,Y 497.887,Z 419.136,A -85,B 0,C 180,E1 22856.776,E2 22856.776} C_VEL
LIN {X 0,Y 497.865,Z 419.336,A -85,B 0,C 180,E1 22855.911,E2 22855.911} C_VEL
LIN {X 0,Y 499.424,Z 423.024,A -85,B 0,C 180,E1 22853.332,E2 22853.332} C_VEL
LIN {X 0,Y 503.164,Z 425.717,A -85,B 0,C 180,E1 22850.044,E2 22850.044} C_VEL
LIN {X 0,Y 504.509,Z 426.254,A -85,B 0,C 180,E1 22849.147,E2 22849.147} C_VEL
LIN {X 0,Y 505.766,Z 429.373,A -85,B 0,C 180,E1 22848.193,E2 22848.193} C_VEL
LIN {X 0,Y 508.559,Z 431.957,A -85,B 0,C 180,E1 22846.585,E2 22846.585} C_VEL
LIN {X 0,Y 510.728,Z 433.127,A -85,B 0,C 180,E1 22845.516,E2 22845.516} C_VEL
LIN {X 0,Y 512.659,Z 436.685,A -85,B 0,C 180,E1 22844.502,E2 22844.502} C_VEL
LIN {X 0,Y 515.659,Z 439.107,A -85,B 0,C 180,E1 22843.207,E2 22843.207} C_VEL
LIN {X 0,Y 516.587,Z 439.779,A -85,B 0,C 180,E1 22842.832,E2 22842.832} C_VEL
LIN {X 0,Y 518.857,Z 443.377,A -85,B 0,C 180,E1 22841.867,E2 22841.867} C_VEL
LIN {X 0,Y 522.327,Z 446.303,A -85,B 0,C 180,E1 22840.602,E2 22840.602} C_VEL
LIN {X 0,Y 525.231,Z 450.298,A -85,B 0,C 180,E1 22839.553,E2 22839.553} C_VEL
LIN {X 0,Y 527.78,Z 452.621,A -85,B 0,C 180,E1 22838.728,E2 22838.728} C_VEL
LIN {X 0,Y 531.145,Z 456.944,A -85,B 0,C 180,E1 22837.65,E2 22837.65} C_VEL
LIN {X 0,Y 533.196,Z 459.018,A -85,B 0,C 180,E1 22837.042,E2 22837.042} C_VEL
LIN {X 0,Y 537.026,Z 463.576,A -85,B 0,C 180,E1 22835.936,E2 22835.936} C_VEL
LIN {X 0,Y 543.362,Z 471.31,A -85,B 0,C 180,E1 22834.231,E2 22834.231} C_VEL
LIN {X 0,Y 548.705,Z 477.887,A -85,B 0,C 180,E1 22832.898,E2 22832.898} C_VEL
LIN {X 0,Y 556.069,Z 487.139,A -85,B 0,C 180,E1 22831.19,E2 22831.19} C_VEL
LIN {X 0,Y 567.388,Z 502.045,A -85,B 0,C 180,E1 22828.794,E2 22828.794} C_VEL
LIN {X 0,Y 580.054,Z 519.796,A -85,B 0,C 180,E1 22826.374,E2 22826.374} C_VEL
LIN {X 0,Y 580.395,Z 520.754,A -85,B 0,C 180,E1 22826.302,E2 22826.302} C_VEL
LIN {X 0,Y 570.928,Z 735.024,A -85,B 0,C 180,E1 22823.085,E2 22823.085} C_VEL
LIN {X 0,Y 564.789,Z 877.521,A -85,B 0,C 180,E1 22820.955,E2 22820.955} C_VEL
LIN {X 0,Y 562.833,Z 902.775,A -85,B 0,C 180,E1 22820.474,E2 22820.474} C_VEL
LIN {X 0,Y 559.834,Z 930.204,A -85,B 0,C 180,E1 22819.761,E2 22819.761} C_VEL
LIN {X 0,Y 556.977,Z 951.628,A -85,B 0,C 180,E1 22819.061,E2 22819.061} C_VEL
LIN {X 0,Y 553.89,Z 971.87,A -85,B 0,C 180,E1 22818.273,E2 22818.273} C_VEL
LIN {X 0,Y 550.419,Z 992.071,A -85,B 0,C 180,E1 22817.358,E2 22817.358} C_VEL
LIN {X 0,Y 546.117,Z 1014.82,A -85,B 0,C 180,E1 22816.158,E2 22816.158} C_VEL
LIN {X 0,Y 540.891,Z 1039.522,A -85,B 0,C 180,E1 22814.615,E2 22814.615} C_VEL
LIN {X 0,Y 538.617,Z 1049.933,A -85,B 0,C 180,E1 22813.89,E2 22813.89} C_VEL
LIN {X 0,Y 536.43,Z 1056.408,A -85,B 0,C 180,E1 22813.496,E2 22813.496} C_VEL
LIN {X 0,Y 527.904,Z 1072.862,A -85,B 0,C 180,E1 22812.642,E2 22812.642} C_VEL
LIN {X 0,Y 525.606,Z 1078.967,A -85,B 0,C 180,E1 22812.192,E2 22812.192} C_VEL
LIN {X 0,Y 519.924,Z 1101.061,A -85,B 0,C 180,E1 22810.1,E2 22810.1} C_VEL
LIN {X 0,Y 514.923,Z 1119.71,A -85,B 0,C 180,E1 22808.054,E2 22808.054} C_VEL
LIN {X 0,Y 510.779,Z 1135.058,A -85,B 0,C 180,E1 22806.163,E2 22806.163} C_VEL
LIN {X 0,Y 506.959,Z 1149.375,A -85,B 0,C 180,E1 22804.194,E2 22804.194} C_VEL
LIN {X 0,Y 502.884,Z 1164.987,A -85,B 0,C 180,E1 22801.788,E2 22801.788} C_VEL
LIN {X 0,Y 498.757,Z 1181.31,A -85,B 0,C 180,E1 22798.883,E2 22798.883} C_VEL
LIN {X 0,Y 495.948,Z 1193.257,A -85,B 0,C 180,E1 22796.452,E2 22796.452} C_VEL
LIN {X 0,Y 493.675,Z 1203.875,A -85,B 0,C 180,E1 22794.012,E2 22794.012} C_VEL
LIN {X 0,Y 491.436,Z 1215.924,A -85,B 0,C 180,E1 22790.851,E2 22790.851} C_VEL
LIN {X 0,Y 489.896,Z 1225.681,A -85,B 0,C 180,E1 22787.821,E2 22787.821} C_VEL
LIN {X 0,Y 489.06,Z 1232.642,A -85,B 0,C 180,E1 22785.286,E2 22785.286} C_VEL
LIN {X 0,Y 488.481,Z 1238.478,A -85,B 0,C 180,E1 22782.766,E2 22782.766} C_VEL
LIN {X 0,Y 488.158,Z 1243.235,A -85,B 0,C 180,E1 22780.259,E2 22780.259} C_VEL
LIN {X 0,Y 487.979,Z 1247.731,A -85,B 0,C 180,E1 22777.174,E2 22777.174} C_VEL
LIN {X 0,Y 487.917,Z 1250.514,A -85,B 0,C 180,E1 22774.107,E2 22774.107} C_VEL
LIN {X 0,Y 487.905,Z 1251.704,A -85,B 0,C 180,E1 22771.521,E2 22771.521} C_VEL
LIN {X 0,Y 487.87,Z 1251.833,A -85,B 0,C 180,E1 22769.055,E2 22769.055} C_VEL
LIN {X 0,Y 487.911,Z 1251.037,A -85,B 0,C 180,E1 22766.705,E2 22766.705} C_VEL
LIN {X 0,Y 487.938,Z 1249.229,A -85,B 0,C 180,E1 22764.232,E2 22764.232} C_VEL
LIN {X 0,Y 488.003,Z 1246.401,A -85,B 0,C 180,E1 22761.747,E2 22761.747} C_VEL
LIN {X 0,Y 488.216,Z 1242.34,A -85,B 0,C 180,E1 22759.135,E2 22759.135} C_VEL
LIN {X 0,Y 488.639,Z 1236.865,A -85,B 0,C 180,E1 22756.385,E2 22756.385} C_VEL
LIN {X 0,Y 489.566,Z 1228.383,A -85,B 0,C 180,E1 22753.014,E2 22753.014} C_VEL
LIN {X 0,Y 490.683,Z 1220.23,A -85,B 0,C 180,E1 22750.348,E2 22750.348} C_VEL
LIN {X 0,Y 492.218,Z 1211.248,A -85,B 0,C 180,E1 22747.796,E2 22747.796} C_VEL
LIN {X 0,Y 494.244,Z 1201.141,A -85,B 0,C 180,E1 22745.238,E2 22745.238} C_VEL
LIN {X 0,Y 497.347,Z 1187.283,A -85,B 0,C 180,E1 22742.193,E2 22742.193} C_VEL
LIN {X 0,Y 500.635,Z 1173.748,A -85,B 0,C 180,E1 22739.634,E2 22739.634} C_VEL
LIN {X 0,Y 503.909,Z 1160.884,A -85,B 0,C 180,E1 22737.466,E2 22737.466} C_VEL
LIN {X 0,Y 507.487,Z 1147.354,A -85,B 0,C 180,E1 22735.424,E2 22735.424} C_VEL
LIN {X 0,Y 512.015,Z 1130.551,A -85,B 0,C 180,E1 22733.16,E2 22733.16} C_VEL
LIN {X 0,Y 517.539,Z 1109.923,A -85,B 0,C 180,E1 22730.751,E2 22730.751} C_VEL
LIN {X 0,Y 522.079,Z 1092.721,A -85,B 0,C 180,E1 22728.99,E2 22728.99} C_VEL
LIN {X 0,Y 526.577,Z 1075.195,A -85,B 0,C 180,E1 22727.391,E2 22727.391} C_VEL
LIN {X 0,Y 531.631,Z 1054.799,A -85,B 0,C 180,E1 22725.748,E2 22725.748} C_VEL
LIN {X 0,Y 537.213,Z 1030.541,A -85,B 0,C 180,E1 22724.07,E2 22724.07} C_VEL
LIN {X 0,Y 541.513,Z 1010.122,A -85,B 0,C 180,E1 22722.854,E2 22722.854} C_VEL
LIN {X 0,Y 545.382,Z 990.105,A -85,B 0,C 180,E1 22721.815,E2 22721.815} C_VEL
LIN {X 0,Y 548.989,Z 969.59,A -85,B 0,C 180,E1 22720.897,E2 22720.897} C_VEL
LIN {X 0,Y 552.955,Z 944.09,A -85,B 0,C 180,E1 22719.936,E2 22719.936} C_VEL
LIN {X 0,Y 556.196,Z 917.876,A -85,B 0,C 180,E1 22719.163,E2 22719.163} C_VEL
LIN {X 0,Y 558.381,Z 896.035,A -85,B 0,C 180,E1 22718.653,E2 22718.653} C_VEL
LIN {X 0,Y 560.028,Z 874.093,A -85,B 0,C 180,E1 22718.256,E2 22718.256} C_VEL
LIN {X 0,Y 569.708,Z 656.791,A -85,B 0,C 180,E1 22714.995,E2 22714.995} C_VEL
LIN {X 0,Y 575.793,Z 524.748,A -85,B 0,C 180,E1 22712.989,E2 22712.989} C_VEL
LIN {X 0,Y 563.793,Z 507.742,A -85,B 0,C 180,E1 22710.627,E2 22710.627} C_VEL
LIN {X 0,Y 552.374,Z 492.576,A -85,B 0,C 180,E1 22708.135,E2 22708.135} C_VEL
LIN {X 0,Y 543.825,Z 481.809,A -85,B 0,C 180,E1 22706.068,E2 22706.068} C_VEL
LIN {X 0,Y 539.132,Z 476.048,A -85,B 0,C 180,E1 22704.839,E2 22704.839} C_VEL
LIN {X 0,Y 534.834,Z 470.784,A -85,B 0,C 180,E1 22703.642,E2 22703.642} C_VEL
LIN {X 0,Y 530.236,Z 465.279,A -85,B 0,C 180,E1 22702.274,E2 22702.274} C_VEL
LIN {X 0,Y 526.515,Z 460.999,A -85,B 0,C 180,E1 22701.093,E2 22701.093} C_VEL
LIN {X 0,Y 525.287,Z 459.388,A -85,B 0,C 180,E1 22700.677,E2 22700.677} C_VEL
LIN {X 0,Y 521.798,Z 455.756,A -85,B 0,C 180,E1 22699.477,E2 22699.477} C_VEL
LIN {X 0,Y 520.129,Z 453.341,A -85,B 0,C 180,E1 22698.842,E2 22698.842} C_VEL
LIN {X 0,Y 516.775,Z 450.307,A -85,B 0,C 180,E1 22697.568,E2 22697.568} C_VEL
LIN {X 0,Y 514.816,Z 447.156,A -85,B 0,C 180,E1 22696.705,E2 22696.705} C_VEL
LIN {X 0,Y 511.338,Z 444.442,A -85,B 0,C 180,E1 22695.191,E2 22695.191} C_VEL
LIN {X 0,Y 509.066,Z 440.581,A -85,B 0,C 180,E1 22693.981,E2 22693.981} C_VEL
LIN {X 0,Y 505.554,Z 438.376,A -85,B 0,C 180,E1 22692.102,E2 22692.102} C_VEL
LIN {X 0,Y 503.596,Z 435.236,A -85,B 0,C 180,E1 22690.757,E2 22690.757} C_VEL
LIN {X 0,Y 503.041,Z 433.896,A -85,B 0,C 180,E1 22690.305,E2 22690.305} C_VEL
LIN {X 0,Y 499.05,Z 431.639,A -85,B 0,C 180,E1 22687.02,E2 22687.02} C_VEL
LIN {X 0,Y 497.032,Z 427.886,A -85,B 0,C 180,E1 22683.922,E2 22683.922} C_VEL
LIN {X 0,Y 496.834,Z 427.06,A -85,B 0,C 180,E1 22683.346,E2 22683.346} C_VEL
LIN {X 0,Y 496.904,Z 427.229,A -85,B 0,C 180,E1 22676.886,E2 22676.886} C_VEL
LIN {X 0,Y 498.702,Z 431.29,A -85,B 0,C 180,E1 22673.784,E2 22673.784} C_VEL
LIN {X 0,Y 502.478,Z 433.727,A -85,B 0,C 180,E1 22670.493,E2 22670.493} C_VEL
LIN {X 0,Y 503.247,Z 434.174,A -85,B 0,C 180,E1 22669.959,E2 22669.959} C_VEL
LIN {X 0,Y 504.862,Z 437.564,A -85,B 0,C 180,E1 22668.75,E2 22668.75} C_VEL
LIN {X 0,Y 507.651,Z 439.986,A -85,B 0,C 180,E1 22667.14,E2 22667.14} C_VEL
LIN {X 0,Y 509.337,Z 441.015,A -85,B 0,C 180,E1 22666.288,E2 22666.288} C_VEL
LIN {X 0,Y 511.475,Z 444.591,A -85,B 0,C 180,E1 22665.162,E2 22665.162} C_VEL
LIN {X 0,Y 515.082,Z 447.539,A -85,B 0,C 180,E1 22663.594,E2 22663.594} C_VEL
LIN {X 0,Y 517.724,Z 451.454,A -85,B 0,C 180,E1 22662.465,E2 22662.465} C_VEL
LIN {X 0,Y 520.258,Z 453.848,A -85,B 0,C 180,E1 22661.511,E2 22661.511} C_VEL
LIN {X 0,Y 524.852,Z 459.628,A -85,B 0,C 180,E1 22659.858,E2 22659.858} C_VEL
LIN {X 0,Y 529.251,Z 465.163,A -85,B 0,C 180,E1 22658.412,E2 22658.412} C_VEL
LIN {X 0,Y 534.184,Z 471.526,A -85,B 0,C 180,E1 22656.912,E2 22656.912} C_VEL
LIN {X 0,Y 541.437,Z 481.193,A -85,B 0,C 180,E1 22654.894,E2 22654.894} C_VEL
LIN {X 0,Y 549.331,Z 492.006,A -85,B 0,C 180,E1 22652.903,E2 22652.903} C_VEL
LIN {X 0,Y 558.588,Z 505.266,A -85,B 0,C 180,E1 22650.775,E2 22650.775} C_VEL
LIN {X 0,Y 569.551,Z 521.846,A -85,B 0,C 180,E1 22648.485,E2 22648.485} C_VEL
LIN {X 0,Y 575.96,Z 532.26,A -85,B 0,C 180,E1 22647.234,E2 22647.234} C_VEL
LIN {X 0,Y 566.158,Z 747.798,A -85,B 0,C 180,E1 22643.982,E2 22643.982} C_VEL
LIN {X 0,Y 559.43,Z 900.431,A -85,B 0,C 180,E1 22641.691,E2 22641.691} C_VEL
LIN {X 0,Y 557.284,Z 926.618,A -85,B 0,C 180,E1 22641.2,E2 22641.2} C_VEL
LIN {X 0,Y 554.077,Z 954.057,A -85,B 0,C 180,E1 22640.499,E2 22640.499} C_VEL
LIN {X 0,Y 551.082,Z 975.507,A -85,B 0,C 180,E1 22639.81,E2 22639.81} C_VEL
LIN {X 0,Y 547.76,Z 996.314,A -85,B 0,C 180,E1 22639.012,E2 22639.012} C_VEL
LIN {X 0,Y 544.13,Z 1016.72,A -85,B 0,C 180,E1 22638.096,E2 22638.096} C_VEL
LIN {X 0,Y 539.395,Z 1041.12,A -85,B 0,C 180,E1 22636.817,E2 22636.817} C_VEL
LIN {X 0,Y 534.031,Z 1065.661,A -85,B 0,C 180,E1 22635.283,E2 22635.283} C_VEL
LIN {X 0,Y 529.5,Z 1085.269,A -85,B 0,C 180,E1 22633.874,E2 22633.874} C_VEL
LIN {X 0,Y 524.997,Z 1103.958,A -85,B 0,C 180,E1 22632.356,E2 22632.356} C_VEL
LIN {X 0,Y 519.606,Z 1125.71,A -85,B 0,C 180,E1 22630.356,E2 22630.356} C_VEL
LIN {X 0,Y 514.378,Z 1146.004,A -85,B 0,C 180,E1 22628.185,E2 22628.185} C_VEL
LIN {X 0,Y 510.241,Z 1162.14,A -85,B 0,C 180,E1 22626.245,E2 22626.245} C_VEL
LIN {X 0,Y 506.475,Z 1177.075,A -85,B 0,C 180,E1 22624.243,E2 22624.243} C_VEL
LIN {X 0,Y 502.331,Z 1193.997,A -85,B 0,C 180,E1 22621.705,E2 22621.705} C_VEL
LIN {X 0,Y 498.512,Z 1210.118,A -85,B 0,C 180,E1 22618.911,E2 22618.911} C_VEL
LIN {X 0,Y 495.796,Z 1222.534,A -85,B 0,C 180,E1 22616.472,E2 22616.472} C_VEL
LIN {X 0,Y 493.702,Z 1233.055,A -85,B 0,C 180,E1 22614.153,E2 22614.153} C_VEL
LIN {X 0,Y 491.928,Z 1242.87,A -85,B 0,C 180,E1 22611.716,E2 22611.716} C_VEL
LIN {X 0,Y 490.273,Z 1253.306,A -85,B 0,C 180,E1 22608.679,E2 22608.679} C_VEL
LIN {X 0,Y 489.159,Z 1261.819,A -85,B 0,C 180,E1 22605.658,E2 22605.658} C_VEL
LIN {X 0,Y 488.527,Z 1268.041,A -85,B 0,C 180,E1 22603.016,E2 22603.016} C_VEL
LIN {X 0,Y 488.187,Z 1272.882,A -85,B 0,C 180,E1 22600.508,E2 22600.508} C_VEL
LIN {X 0,Y 487.978,Z 1276.821,A -85,B 0,C 180,E1 22597.896,E2 22597.896} C_VEL
LIN {X 0,Y 487.925,Z 1279.868,A -85,B 0,C 180,E1 22595.06,E2 22595.06} C_VEL
LIN {X 0,Y 487.909,Z 1281.643,A -85,B 0,C 180,E1 22591.884,E2 22591.884} C_VEL
LIN {X 0,Y 487.865,Z 1281.872,A -85,B 0,C 180,E1 22589.301,E2 22589.301} C_VEL
LIN {X 0,Y 487.91,Z 1281.084,A -85,B 0,C 180,E1 22586.834,E2 22586.834} C_VEL
LIN {X 0,Y 487.934,Z 1279.309,A -85,B 0,C 180,E1 22584.361,E2 22584.361} C_VEL
LIN {X 0,Y 487.994,Z 1276.515,A -85,B 0,C 180,E1 22581.878,E2 22581.878} C_VEL
LIN {X 0,Y 488.212,Z 1272.487,A -85,B 0,C 180,E1 22579.265,E2 22579.265} C_VEL
LIN {X 0,Y 488.602,Z 1267.301,A -85,B 0,C 180,E1 22576.636,E2 22576.636} C_VEL
LIN {X 0,Y 489.462,Z 1259.244,A -85,B 0,C 180,E1 22573.354,E2 22573.354} C_VEL
LIN {X 0,Y 490.637,Z 1250.524,A -85,B 0,C 180,E1 22570.482,E2 22570.482} C_VEL
LIN {X 0,Y 492.077,Z 1241.99,A -85,B 0,C 180,E1 22568.052,E2 22568.052} C_VEL
LIN {X 0,Y 493.898,Z 1232.058,A -85,B 0,C 180,E1 22565.614,E2 22565.614} C_VEL
LIN {X 0,Y 496.175,Z 1220.839,A -85,B 0,C 180,E1 22563.174,E2 22563.174} C_VEL
LIN {X 0,Y 499.575,Z 1205.553,A -85,B 0,C 180,E1 22560.248,E2 22560.248} C_VEL
LIN {X 0,Y 503.228,Z 1190.15,A -85,B 0,C 180,E1 22557.699,E2 22557.699} C_VEL
LIN {X 0,Y 506.825,Z 1175.631,A -85,B 0,C 180,E1 22555.554,E2 22555.554} C_VEL
LIN {X 0,Y 510.777,Z 1160.048,A -85,B 0,C 180,E1 22553.489,E2 22553.489} C_VEL
LIN {X 0,Y 515.996,Z 1139.85,A -85,B 0,C 180,E1 22551.118,E2 22551.118} C_VEL
LIN {X 0,Y 520.945,Z 1120.257,A -85,B 0,C 180,E1 22549.127,E2 22549.127} C_VEL
LIN {X 0,Y 525.389,Z 1102.34,A -85,B 0,C 180,E1 22547.508,E2 22547.508} C_VEL
LIN {X 0,Y 529.826,Z 1083.897,A -85,B 0,C 180,E1 22546.024,E2 22546.024} C_VEL
LIN {X 0,Y 534.805,Z 1062.354,A -85,B 0,C 180,E1 22544.495,E2 22544.495} C_VEL
LIN {X 0,Y 540.22,Z 1036.888,A -85,B 0,C 180,E1 22542.954,E2 22542.954} C_VEL
LIN {X 0,Y 544.294,Z 1015.75,A -85,B 0,C 180,E1 22541.859,E2 22541.859} C_VEL
LIN {X 0,Y 547.931,Z 995.2,A -85,B 0,C 180,E1 22540.943,E2 22540.943} C_VEL
LIN {X 0,Y 551.259,Z 974.219,A -85,B 0,C 180,E1 22540.146,E2 22540.146} C_VEL
LIN {X 0,Y 554.862,Z 948.297,A -85,B 0,C 180,E1 22539.334,E2 22539.334} C_VEL
LIN {X 0,Y 557.711,Z 921.572,A -85,B 0,C 180,E1 22538.7,E2 22538.7} C_VEL
LIN {X 0,Y 559.503,Z 898.806,A -85,B 0,C 180,E1 22538.285,E2 22538.285} C_VEL
LIN {X 0,Y 568.796,Z 687.393,A -85,B 0,C 180,E1 22535.114,E2 22535.114} C_VEL
LIN {X 0,Y 575.869,Z 532.039,A -85,B 0,C 180,E1 22532.757,E2 22532.757} C_VEL
LIN {X 0,Y 565.578,Z 515.796,A -85,B 0,C 180,E1 22530.726,E2 22530.726} C_VEL
LIN {X 0,Y 556.715,Z 502.692,A -85,B 0,C 180,E1 22528.832,E2 22528.832} C_VEL
LIN {X 0,Y 547.772,Z 489.812,A -85,B 0,C 180,E1 22526.741,E2 22526.741} C_VEL
LIN {X 0,Y 538.768,Z 477.668,A -85,B 0,C 180,E1 22524.419,E2 22524.419} C_VEL
LIN {X 0,Y 532.029,Z 468.789,A -85,B 0,C 180,E1 22522.486,E2 22522.486} C_VEL
LIN {X 0,Y 527.607,Z 463.129,A -85,B 0,C 180,E1 22521.105,E2 22521.105} C_VEL
LIN {X 0,Y 523.147,Z 457.548,A -85,B 0,C 180,E1 22519.599,E2 22519.599} C_VEL
LIN {X 0,Y 519.267,Z 452.843,A -85,B 0,C 180,E1 22518.176,E2 22518.176} C_VEL
LIN {X 0,Y 516.137,Z 449.53,A -85,B 0,C 180,E1 22516.951,E2 22516.951} C_VEL
LIN {X 0,Y 514.813,Z 447.182,A -85,B 0,C 180,E1 22516.357,E2 22516.357} C_VEL
LIN {X 0,Y 511.428,Z 444.575,A -85,B 0,C 180,E1 22514.898,E2 22514.898} C_VEL
LIN {X 0,Y 509.215,Z 440.969,A -85,B 0,C 180,E1 22513.745,E2 22513.745} C_VEL
LIN {X 0,Y 507.897,Z 440.133,A -85,B 0,C 180,E1 22513.085,E2 22513.085} C_VEL
LIN {X 0,Y 504.934,Z 437.755,A -85,B 0,C 180,E1 22511.421,E2 22511.421} C_VEL
LIN {X 0,Y 503.13,Z 434.101,A -85,B 0,C 180,E1 22510.101,E2 22510.101} C_VEL
LIN {X 0,Y 498.577,Z 431.258,A -85,B 0,C 180,E1 22506.333,E2 22506.333} C_VEL
LIN {X 0,Y 496.861,Z 427.47,A -85,B 0,C 180,E1 22503.577,E2 22503.577} C_VEL
LIN {X 0,Y 496.663,Z 427.042,A -85,B 0,C 180,E1 22503.116,E2 22503.116} C_VEL
LIN {X 0,Y 496.81,Z 427.145,A -85,B 0,C 180,E1 22496.076,E2 22496.076} C_VEL
LIN {X 0,Y 498.353,Z 430.903,A -85,B 0,C 180,E1 22493.433,E2 22493.433} C_VEL
LIN {X 0,Y 502.041,Z 433.611,A -85,B 0,C 180,E1 22490.138,E2 22490.138} C_VEL
LIN {X 0,Y 503.227,Z 434.228,A -85,B 0,C 180,E1 22489.322,E2 22489.322} C_VEL
LIN {X 0,Y 504.696,Z 437.439,A -85,B 0,C 180,E1 22488.225,E2 22488.225} C_VEL
LIN {X 0,Y 507.818,Z 440.083,A -85,B 0,C 180,E1 22486.449,E2 22486.449} C_VEL
LIN {X 0,Y 509.305,Z 440.985,A -85,B 0,C 180,E1 22485.707,E2 22485.707} C_VEL
LIN {X 0,Y 511.454,Z 444.653,A -85,B 0,C 180,E1 22484.581,E2 22484.581} C_VEL
LIN {X 0,Y 515.025,Z 447.548,A -85,B 0,C 180,E1 22483.04,E2 22483.04} C_VEL
LIN {X 0,Y 517.619,Z 451.362,A -85,B 0,C 180,E1 22481.938,E2 22481.938} C_VEL
LIN {X 0,Y 520.626,Z 453.946,A -85,B 0,C 180,E1 22480.827,E2 22480.827} C_VEL
LIN {X 0,Y 523.812,Z 458.143,A -85,B 0,C 180,E1 22479.671,E2 22479.671} C_VEL
LIN {X 0,Y 526.011,Z 460.272,A -85,B 0,C 180,E1 22478.945,E2 22478.945} C_VEL
LIN {X 0,Y 529.52,Z 464.646,A -85,B 0,C 180,E1 22477.811,E2 22477.811} C_VEL
LIN {X 0,Y 531.288,Z 466.541,A -85,B 0,C 180,E1 22477.276,E2 22477.276} C_VEL
LIN {X 0,Y 535.357,Z 471.279,A -85,B 0,C 180,E1 22476.09,E2 22476.09} C_VEL
LIN {X 0,Y 540.064,Z 477.034,A -85,B 0,C 180,E1 22474.797,E2 22474.797} C_VEL
LIN {X 0,Y 549.54,Z 489.025,A -85,B 0,C 180,E1 22472.415,E2 22472.415} C_VEL
LIN {X 0,Y 560.655,Z 503.537,A -85,B 0,C 180,E1 22469.924,E2 22469.924} C_VEL
LIN {X 0,Y 572.456,Z 519.97,A -85,B 0,C 180,E1 22467.543,E2 22467.543} C_VEL
LIN {X 0,Y 575.796,Z 525.107,A -85,B 0,C 180,E1 22466.903,E2 22466.903} C_VEL
LIN {X 0,Y 565.952,Z 739.861,A -85,B 0,C 180,E1 22463.665,E2 22463.665} C_VEL
LIN {X 0,Y 559.779,Z 877.841,A -85,B 0,C 180,E1 22461.591,E2 22461.591} C_VEL
LIN {X 0,Y 557.737,Z 903.404,A -85,B 0,C 180,E1 22461.101,E2 22461.101} C_VEL
LIN {X 0,Y 554.647,Z 930.697,A -85,B 0,C 180,E1 22460.388,E2 22460.388} C_VEL
LIN {X 0,Y 551.679,Z 952.251,A -85,B 0,C 180,E1 22459.681,E2 22459.681} C_VEL
LIN {X 0,Y 548.544,Z 972.145,A -85,B 0,C 180,E1 22458.903,E2 22458.903} C_VEL
LIN {X 0,Y 544.955,Z 992.346,A -85,B 0,C 180,E1 22457.985,E2 22457.985} C_VEL
LIN {X 0,Y 540.509,Z 1015.096,A -85,B 0,C 180,E1 22456.78,E2 22456.78} C_VEL
LIN {X 0,Y 534.998,Z 1040.205,A -85,B 0,C 180,E1 22455.203,E2 22455.203} C_VEL
LIN {X 0,Y 530.526,Z 1059.121,A -85,B 0,C 180,E1 22453.829,E2 22453.829} C_VEL
LIN {X 0,Y 526.068,Z 1077.131,A -85,B 0,C 180,E1 22452.351,E2 22452.351} C_VEL
LIN {X 0,Y 525.606,Z 1078.967,A -85,B 0,C 180,E1 22452.192,E2 22452.192} C_VEL
LIN {X 0,Y 523.325,Z 1085.093,A -85,B 0,C 180,E1 22451.729,E2 22451.729} C_VEL
LIN {X 0,Y 514.569,Z 1100.671,A -85,B 0,C 180,E1 22450.691,E2 22450.691} C_VEL
LIN {X 0,Y 512.232,Z 1106.263,A -85,B 0,C 180,E1 22450.167,E2 22450.167} C_VEL
LIN {X 0,Y 507.889,Z 1121.823,A -85,B 0,C 180,E1 22448.413,E2 22448.413} C_VEL
LIN {X 0,Y 503.541,Z 1137.281,A -85,B 0,C 180,E1 22446.465,E2 22446.465} C_VEL
LIN {X 0,Y 498.523,Z 1155.427,A -85,B 0,C 180,E1 22443.88,E2 22443.88} C_VEL
LIN {X 0,Y 494.251,Z 1170.927,A -85,B 0,C 180,E1 22441.319,E2 22441.319} C_VEL
LIN {X 0,Y 490.994,Z 1183.455,A -85,B 0,C 180,E1 22438.983,E2 22438.983} C_VEL
LIN {X 0,Y 488.239,Z 1194.657,A -85,B 0,C 180,E1 22436.64,E2 22436.64} C_VEL
LIN {X 0,Y 485.681,Z 1206.149,A -85,B 0,C 180,E1 22433.92,E2 22433.92} C_VEL
LIN {X 0,Y 483.393,Z 1217.721,A -85,B 0,C 180,E1 22430.707,E2 22430.707} C_VEL
LIN {X 0,Y 481.939,Z 1226.388,A -85,B 0,C 180,E1 22427.875,E2 22427.875} C_VEL
LIN {X 0,Y 481.089,Z 1233.15,A -85,B 0,C 180,E1 22425.339,E2 22425.339} C_VEL
LIN {X 0,Y 480.462,Z 1239.242,A -85,B 0,C 180,E1 22422.616,E2 22422.616} C_VEL
LIN {X 0,Y 480.063,Z 1244.852,A -85,B 0,C 180,E1 22419.465,E2 22419.465} C_VEL
LIN {X 0,Y 479.959,Z 1248.614,A -85,B 0,C 180,E1 22416.419,E2 22416.419} C_VEL
LIN {X 0,Y 479.914,Z 1250.718,A -85,B 0,C 180,E1 22413.817,E2 22413.817} C_VEL
LIN {X 0,Y 479.903,Z 1251.727,A -85,B 0,C 180,E1 22411.427,E2 22411.427} C_VEL
LIN {X 0,Y 479.871,Z 1251.833,A -85,B 0,C 180,E1 22409.039,E2 22409.039} C_VEL
LIN {X 0,Y 479.911,Z 1251.036,A -85,B 0,C 180,E1 22406.65,E2 22406.65} C_VEL
LIN {X 0,Y 479.942,Z 1249.226,A -85,B 0,C 180,E1 22404.136,E2 22404.136} C_VEL
LIN {X 0,Y 480.019,Z 1246.399,A -85,B 0,C 180,E1 22401.611,E2 22401.611} C_VEL
LIN {X 0,Y 480.235,Z 1242.335,A -85,B 0,C 180,E1 22398.952,E2 22398.952} C_VEL
LIN {X 0,Y 480.666,Z 1237.117,A -85,B 0,C 180,E1 22396.277,E2 22396.277} C_VEL
LIN {X 0,Y 481.644,Z 1228.733,A -85,B 0,C 180,E1 22392.85,E2 22392.85} C_VEL
LIN {X 0,Y 482.968,Z 1219.943,A -85,B 0,C 180,E1 22389.895,E2 22389.895} C_VEL
LIN {X 0,Y 484.543,Z 1211.518,A -85,B 0,C 180,E1 22387.425,E2 22387.425} C_VEL
LIN {X 0,Y 486.702,Z 1201.411,A -85,B 0,C 180,E1 22384.828,E2 22384.828} C_VEL
LIN {X 0,Y 489.988,Z 1187.552,A -85,B 0,C 180,E1 22381.739,E2 22381.739} C_VEL
LIN {X 0,Y 493.435,Z 1174.071,A -85,B 0,C 180,E1 22379.154,E2 22379.154} C_VEL
LIN {X 0,Y 496.879,Z 1161.154,A -85,B 0,C 180,E1 22376.948,E2 22376.948} C_VEL
LIN {X 0,Y 500.633,Z 1147.623,A -85,B 0,C 180,E1 22374.882,E2 22374.882} C_VEL
LIN {X 0,Y 505.374,Z 1130.819,A -85,B 0,C 180,E1 22372.594,E2 22372.594} C_VEL
LIN {X 0,Y 511.013,Z 1110.683,A -85,B 0,C 180,E1 22370.217,E2 22370.217} C_VEL
LIN {X 0,Y 515.682,Z 1093.689,A -85,B 0,C 180,E1 22368.456,E2 22368.456} C_VEL
LIN {X 0,Y 520.193,Z 1076.781,A -85,B 0,C 180,E1 22366.892,E2 22366.892} C_VEL
LIN {X 0,Y 524.757,Z 1058.989,A -85,B 0,C 180,E1 22365.427,E2 22365.427} C_VEL
LIN {X 0,Y 529.975,Z 1037.678,A -85,B 0,C 180,E1 22363.883,E2 22363.883} C_VEL
LIN {X 0,Y 535.462,Z 1013.029,A -85,B 0,C 180,E1 22362.362,E2 22362.362} C_VEL
LIN {X 0,Y 539.611,Z 992.444,A -85,B 0,C 180,E1 22361.274,E2 22361.274} C_VEL
LIN {X 0,Y 543.289,Z 972.398,A -85,B 0,C 180,E1 22360.361,E2 22360.361} C_VEL
LIN {X 0,Y 546.672,Z 951.591,A -85,B 0,C 180,E1 22359.55,E2 22359.55} C_VEL
LIN {X 0,Y 550.051,Z 927.569,A -85,B 0,C 180,E1 22358.771,E2 22358.771} C_VEL
LIN {X 0,Y 553.105,Z 899.678,A -85,B 0,C 180,E1 22358.075,E2 22358.075} C_VEL
LIN {X 0,Y 554.95,Z 876.815,A -85,B 0,C 180,E1 22357.648,E2 22357.648} C_VEL
LIN {X 0,Y 564.529,Z 670.217,A -85,B 0,C 180,E1 22354.529,E2 22354.529} C_VEL
LIN {X 0,Y 571.285,Z 529.215,A -85,B 0,C 180,E1 22352.383,E2 22352.383} C_VEL
LIN {X 0,Y 559.95,Z 513.195,A -85,B 0,C 180,E1 22350.088,E2 22350.088} C_VEL
LIN {X 0,Y 549.66,Z 499.356,A -85,B 0,C 180,E1 22347.785,E2 22347.785} C_VEL
LIN {X 0,Y 541.324,Z 488.749,A -85,B 0,C 180,E1 22345.726,E2 22345.726} C_VEL
LIN {X 0,Y 536.699,Z 483.012,A -85,B 0,C 180,E1 22344.49,E2 22344.49} C_VEL
LIN {X 0,Y 532.641,Z 477.981,A -85,B 0,C 180,E1 22343.334,E2 22343.334} C_VEL
LIN {X 0,Y 528.274,Z 472.682,A -85,B 0,C 180,E1 22342.01,E2 22342.01} C_VEL
LIN {X 0,Y 524.457,Z 468.141,A -85,B 0,C 180,E1 22340.77,E2 22340.77} C_VEL
LIN {X 0,Y 523.073,Z 466.584,A -85,B 0,C 180,E1 22340.301,E2 22340.301} C_VEL
LIN {X 0,Y 519.549,Z 462.487,A -85,B 0,C 180,E1 22339.039,E2 22339.039} C_VEL
LIN {X 0,Y 518.597,Z 461.049,A -85,B 0,C 180,E1 22338.667,E2 22338.667} C_VEL
LIN {X 0,Y 515.151,Z 457.851,A -85,B 0,C 180,E1 22337.334,E2 22337.334} C_VEL
LIN {X 0,Y 513.076,Z 454.762,A -85,B 0,C 180,E1 22336.414,E2 22336.414} C_VEL
LIN {X 0,Y 509.692,Z 451.854,A -85,B 0,C 180,E1 22334.892,E2 22334.892} C_VEL
LIN {X 0,Y 507.663,Z 448.387,A -85,B 0,C 180,E1 22333.788,E2 22333.788} C_VEL
LIN {X 0,Y 504.22,Z 446.079,A -85,B 0,C 180,E1 22331.902,E2 22331.902} C_VEL
LIN {X 0,Y 502.234,Z 442.783,A -85,B 0,C 180,E1 22330.496,E2 22330.496} C_VEL
LIN {X 0,Y 501.745,Z 441.753,A -85,B 0,C 180,E1 22330.1,E2 22330.1} C_VEL
LIN {X 0,Y 497.768,Z 439.313,A -85,B 0,C 180,E1 22326.691,E2 22326.691} C_VEL
LIN {X 0,Y 495.963,Z 435.588,A -85,B 0,C 180,E1 22323.699,E2 22323.699} C_VEL
LIN {X 0,Y 495.757,Z 434.984,A -85,B 0,C 180,E1 22323.122,E2 22323.122} C_VEL
LIN {X 0,Y 495.877,Z 435.142,A -85,B 0,C 180,E1 22316.995,E2 22316.995} C_VEL
LIN {X 0,Y 497.727,Z 439.278,A -85,B 0,C 180,E1 22313.772,E2 22313.772} C_VEL
LIN {X 0,Y 501.679,Z 441.728,A -85,B 0,C 180,E1 22310.362,E2 22310.362} C_VEL
LIN {X 0,Y 502.116,Z 442.427,A -85,B 0,C 180,E1 22310.023,E2 22310.023} C_VEL
LIN {X 0,Y 504.055,Z 445.926,A -85,B 0,C 180,E1 22308.616,E2 22308.616} C_VEL
LIN {X 0,Y 507.347,Z 448.276,A -85,B 0,C 180,E1 22306.784,E2 22306.784} C_VEL
LIN {X 0,Y 508.021,Z 449.031,A -85,B 0,C 180,E1 22306.426,E2 22306.426} C_VEL
LIN {X 0,Y 510.502,Z 452.785,A -85,B 0,C 180,E1 22305.133,E2 22305.133} C_VEL
LIN {X 0,Y 513.532,Z 455.265,A -85,B 0,C 180,E1 22303.804,E2 22303.804} C_VEL
LIN {X 0,Y 516.351,Z 459.281,A -85,B 0,C 180,E1 22302.591,E2 22302.591} C_VEL
LIN {X 0,Y 518.581,Z 461.405,A -85,B 0,C 180,E1 22301.74,E2 22301.74} C_VEL
LIN {X 0,Y 523.112,Z 467.215,A -85,B 0,C 180,E1 22300.08,E2 22300.08} C_VEL
LIN {X 0,Y 527.379,Z 472.656,A -85,B 0,C 180,E1 22298.652,E2 22298.652} C_VEL
LIN {X 0,Y 532.254,Z 479.025,A -85,B 0,C 180,E1 22297.145,E2 22297.145} C_VEL
LIN {X 0,Y 539.243,Z 488.474,A -85,B 0,C 180,E1 22295.166,E2 22295.166} C_VEL
LIN {X 0,Y 547.343,Z 499.734,A -85,B 0,C 180,E1 22293.09,E2 22293.09} C_VEL
LIN {X 0,Y 556.311,Z 512.8,A -85,B 0,C 180,E1 22290.998,E2 22290.998} C_VEL
LIN {X 0,Y 566.729,Z 528.786,A -85,B 0,C 180,E1 22288.784,E2 22288.784} C_VEL
LIN {X 0,Y 571.412,Z 536.547,A -85,B 0,C 180,E1 22287.845,E2 22287.845} C_VEL
LIN {X 0,Y 561.301,Z 751.022,A -85,B 0,C 180,E1 22284.595,E2 22284.595} C_VEL
LIN {X 0,Y 554.475,Z 900.184,A -85,B 0,C 180,E1 22282.343,E2 22282.343} C_VEL
LIN {X 0,Y 552.254,Z 926.53,A -85,B 0,C 180,E1 22281.849,E2 22281.849} C_VEL
LIN {X 0,Y 548.966,Z 953.8,A -85,B 0,C 180,E1 22281.151,E2 22281.151} C_VEL
LIN {X 0,Y 545.869,Z 975.248,A -85,B 0,C 180,E1 22280.462,E2 22280.462} C_VEL
LIN {X 0,Y 542.441,Z 996.051,A -85,B 0,C 180,E1 22279.663,E2 22279.663} C_VEL
LIN {X 0,Y 538.687,Z 1016.457,A -85,B 0,C 180,E1 22278.745,E2 22278.745} C_VEL
LIN {X 0,Y 533.732,Z 1041.159,A -85,B 0,C 180,E1 22277.445,E2 22277.445} C_VEL
LIN {X 0,Y 528.235,Z 1065.392,A -85,B 0,C 180,E1 22275.922,E2 22275.922} C_VEL
LIN {X 0,Y 523.537,Z 1085,A -85,B 0,C 180,E1 22274.505,E2 22274.505} C_VEL
LIN {X 0,Y 518.948,Z 1103.312,A -85,B 0,C 180,E1 22273.01,E2 22273.01} C_VEL
LIN {X 0,Y 513.65,Z 1123.821,A -85,B 0,C 180,E1 22271.118,E2 22271.118} C_VEL
LIN {X 0,Y 507.959,Z 1145.01,A -85,B 0,C 180,E1 22268.858,E2 22268.858} C_VEL
LIN {X 0,Y 503.527,Z 1161.563,A -85,B 0,C 180,E1 22266.853,E2 22266.853} C_VEL
LIN {X 0,Y 499.494,Z 1176.797,A -85,B 0,C 180,E1 22264.79,E2 22264.79} C_VEL
LIN {X 0,Y 495.146,Z 1193.795,A -85,B 0,C 180,E1 22262.207,E2 22262.207} C_VEL
LIN {X 0,Y 491.111,Z 1209.893,A -85,B 0,C 180,E1 22259.378,E2 22259.378} C_VEL
LIN {X 0,Y 488.284,Z 1222.258,A -85,B 0,C 180,E1 22256.912,E2 22256.912} C_VEL
LIN {X 0,Y 485.955,Z 1233.305,A -85,B 0,C 180,E1 22254.434,E2 22254.434} C_VEL
LIN {X 0,Y 483.726,Z 1245.418,A -85,B 0,C 180,E1 22251.338,E2 22251.338} C_VEL
LIN {X 0,Y 482.151,Z 1255.073,A -85,B 0,C 180,E1 22248.379,E2 22248.379} C_VEL
LIN {X 0,Y 481.18,Z 1262.425,A -85,B 0,C 180,E1 22245.677,E2 22245.677} C_VEL
LIN {X 0,Y 480.556,Z 1268.295,A -85,B 0,C 180,E1 22243.113,E2 22243.113} C_VEL
LIN {X 0,Y 480.198,Z 1273.085,A -85,B 0,C 180,E1 22240.563,E2 22240.563} C_VEL
LIN {X 0,Y 479.972,Z 1277.298,A -85,B 0,C 180,E1 22237.667,E2 22237.667} C_VEL
LIN {X 0,Y 479.92,Z 1280.33,A -85,B 0,C 180,E1 22234.546,E2 22234.546} C_VEL
LIN {X 0,Y 479.906,Z 1281.688,A -85,B 0,C 180,E1 22231.677,E2 22231.677} C_VEL
LIN {X 0,Y 479.867,Z 1281.849,A -85,B 0,C 180,E1 22229.17,E2 22229.17} C_VEL
LIN {X 0,Y 479.91,Z 1281.016,A -85,B 0,C 180,E1 22226.661,E2 22226.661} C_VEL
LIN {X 0,Y 479.941,Z 1279.193,A -85,B 0,C 180,E1 22224.147,E2 22224.147} C_VEL
LIN {X 0,Y 480.014,Z 1276.416,A -85,B 0,C 180,E1 22221.67,E2 22221.67} C_VEL
LIN {X 0,Y 480.231,Z 1272.484,A -85,B 0,C 180,E1 22219.084,E2 22219.084} C_VEL
LIN {X 0,Y 480.63,Z 1267.555,A -85,B 0,C 180,E1 22216.533,E2 22216.533} C_VEL
LIN {X 0,Y 481.48,Z 1260.025,A -85,B 0,C 180,E1 22213.353,E2 22213.353} C_VEL
LIN {X 0,Y 482.702,Z 1251.271,A -85,B 0,C 180,E1 22210.4,E2 22210.4} C_VEL
LIN {X 0,Y 484.251,Z 1242.185,A -85,B 0,C 180,E1 22207.806,E2 22207.806} C_VEL
LIN {X 0,Y 486.156,Z 1232.309,A -85,B 0,C 180,E1 22205.33,E2 22205.33} C_VEL
LIN {X 0,Y 488.543,Z 1221.148,A -85,B 0,C 180,E1 22202.852,E2 22202.852} C_VEL
LIN {X 0,Y 491.978,Z 1206.492,A -85,B 0,C 180,E1 22199.974,E2 22199.974} C_VEL
LIN {X 0,Y 496.087,Z 1189.872,A -85,B 0,C 180,E1 22197.176,E2 22197.176} C_VEL
LIN {X 0,Y 499.691,Z 1176.017,A -85,B 0,C 180,E1 22195.099,E2 22195.099} C_VEL
LIN {X 0,Y 503.753,Z 1160.71,A -85,B 0,C 180,E1 22193.037,E2 22193.037} C_VEL
LIN {X 0,Y 508.739,Z 1142.223,A -85,B 0,C 180,E1 22190.82,E2 22190.82} C_VEL
LIN {X 0,Y 514.458,Z 1120.656,A -85,B 0,C 180,E1 22188.581,E2 22188.581} C_VEL
LIN {X 0,Y 519.087,Z 1102.738,A -85,B 0,C 180,E1 22186.943,E2 22186.943} C_VEL
LIN {X 0,Y 523.499,Z 1085.105,A -85,B 0,C 180,E1 22185.505,E2 22185.505} C_VEL
LIN {X 0,Y 528.194,Z 1065.509,A -85,B 0,C 180,E1 22184.088,E2 22184.088} C_VEL
LIN {X 0,Y 533.721,Z 1041.152,A -85,B 0,C 180,E1 22182.556,E2 22182.556} C_VEL
LIN {X 0,Y 538.641,Z 1016.613,A -85,B 0,C 180,E1 22181.264,E2 22181.264} C_VEL
LIN {X 0,Y 542.391,Z 996.217,A -85,B 0,C 180,E1 22180.346,E2 22180.346} C_VEL
LIN {X 0,Y 545.818,Z 975.432,A -85,B 0,C 180,E1 22179.547,E2 22179.547} C_VEL
LIN {X 0,Y 549.051,Z 953.032,A -85,B 0,C 180,E1 22178.828,E2 22178.828} C_VEL
LIN {X 0,Y 552.419,Z 924.444,A -85,B 0,C 180,E1 22178.111,E2 22178.111} C_VEL
LIN {X 0,Y 554.476,Z 899.706,A -85,B 0,C 180,E1 22177.651,E2 22177.651} C_VEL
LIN {X 0,Y 563.783,Z 696.023,A -85,B 0,C 180,E1 22174.578,E2 22174.578} C_VEL
LIN {X 0,Y 571.31,Z 536.281,A -85,B 0,C 180,E1 22172.144,E2 22172.144} C_VEL
LIN {X 0,Y 560.299,Z 518.833,A -85,B 0,C 180,E1 22169.89,E2 22169.89} C_VEL
LIN {X 0,Y 548.956,Z 502.037,A -85,B 0,C 180,E1 22167.323,E2 22167.323} C_VEL
LIN {X 0,Y 540.067,Z 489.704,A -85,B 0,C 180,E1 22165.086,E2 22165.086} C_VEL
LIN {X 0,Y 533.787,Z 481.073,A -85,B 0,C 180,E1 22163.34,E2 22163.34} C_VEL
LIN {X 0,Y 529.367,Z 475.377,A -85,B 0,C 180,E1 22162.02,E2 22162.02} C_VEL
LIN {X 0,Y 525.676,Z 470.502,A -85,B 0,C 180,E1 22160.836,E2 22160.836} C_VEL
LIN {X 0,Y 520.841,Z 464.407,A -85,B 0,C 180,E1 22159.164,E2 22159.164} C_VEL
LIN {X 0,Y 517.596,Z 460.431,A -85,B 0,C 180,E1 22157.946,E2 22157.946} C_VEL
LIN {X 0,Y 514.392,Z 456.89,A -85,B 0,C 180,E1 22156.661,E2 22156.661} C_VEL
LIN {X 0,Y 513.066,Z 454.794,A -85,B 0,C 180,E1 22156.066,E2 22156.066} C_VEL
LIN {X 0,Y 509.77,Z 451.995,A -85,B 0,C 180,E1 22154.599,E2 22154.599} C_VEL
LIN {X 0,Y 507.386,Z 448.303,A -85,B 0,C 180,E1 22153.331,E2 22153.331} C_VEL
LIN {X 0,Y 504.044,Z 446,A -85,B 0,C 180,E1 22151.5,E2 22151.5} C_VEL
LIN {X 0,Y 501.932,Z 442.164,A -85,B 0,C 180,E1 22149.98,E2 22149.98} C_VEL
LIN {X 0,Y 501.301,Z 441.633,A -85,B 0,C 180,E1 22149.529,E2 22149.529} C_VEL
LIN {X 0,Y 497.501,Z 439.136,A -85,B 0,C 180,E1 22146.231,E2 22146.231} C_VEL
LIN {X 0,Y 495.807,Z 435.276,A -85,B 0,C 180,E1 22143.411,E2 22143.411} C_VEL
LIN {X 0,Y 495.104,Z 434.903,A -85,B 0,C 180,E1 22141.62,E2 22141.62} C_VEL
LIN {X 0,Y 495.795,Z 435.172,A -85,B 0,C 180,E1 22136.126,E2 22136.126} C_VEL
LIN {X 0,Y 497.282,Z 438.782,A -85,B 0,C 180,E1 22133.535,E2 22133.535} C_VEL
LIN {X 0,Y 500.92,Z 441.504,A -85,B 0,C 180,E1 22130.231,E2 22130.231} C_VEL
LIN {X 0,Y 501.96,Z 442.125,A -85,B 0,C 180,E1 22129.498,E2 22129.498} C_VEL
LIN {X 0,Y 503.63,Z 445.477,A -85,B 0,C 180,E1 22128.258,E2 22128.258} C_VEL
LIN {X 0,Y 507.083,Z 448.178,A -85,B 0,C 180,E1 22126.313,E2 22126.313} C_VEL
LIN {X 0,Y 507.893,Z 448.803,A -85,B 0,C 180,E1 22125.899,E2 22125.899} C_VEL
LIN {X 0,Y 510.252,Z 452.602,A -85,B 0,C 180,E1 22124.66,E2 22124.66} C_VEL
LIN {X 0,Y 513.474,Z 455.274,A -85,B 0,C 180,E1 22123.25,E2 22123.25} C_VEL
LIN {X 0,Y 516.247,Z 459.192,A -85,B 0,C 180,E1 22122.064,E2 22122.064} C_VEL
LIN {X 0,Y 518.936,Z 461.563,A -85,B 0,C 180,E1 22121.054,E2 22121.054} C_VEL
LIN {X 0,Y 522.242,Z 465.837,A -85,B 0,C 180,E1 22119.841,E2 22119.841} C_VEL
LIN {X 0,Y 524.254,Z 467.9,A -85,B 0,C 180,E1 22119.163,E2 22119.163} C_VEL
LIN {X 0,Y 528.068,Z 472.498,A -85,B 0,C 180,E1 22117.923,E2 22117.923} C_VEL
LIN {X 0,Y 534.362,Z 480.146,A -85,B 0,C 180,E1 22116.043,E2 22116.043} C_VEL
LIN {X 0,Y 539.344,Z 486.371,A -85,B 0,C 180,E1 22114.673,E2 22114.673} C_VEL
LIN {X 0,Y 546.574,Z 495.327,A -85,B 0,C 180,E1 22112.843,E2 22112.843} C_VEL
LIN {X 0,Y 558.261,Z 510.905,A -85,B 0,C 180,E1 22110.167,E2 22110.167} C_VEL
LIN {X 0,Y 569.387,Z 526.538,A -85,B 0,C 180,E1 22107.883,E2 22107.883} C_VEL
LIN {X 0,Y 571.262,Z 529.451,A -85,B 0,C 180,E1 22107.514,E2 22107.514} C_VEL
LIN {X 0,Y 561.032,Z 744.781,A -85,B 0,C 180,E1 22104.254,E2 22104.254} C_VEL
LIN {X 0,Y 554.839,Z 878.157,A -85,B 0,C 180,E1 22102.238,E2 22102.238} C_VEL
LIN {X 0,Y 552.709,Z 904.028,A -85,B 0,C 180,E1 22101.741,E2 22101.741} C_VEL
LIN {X 0,Y 549.527,Z 931.189,A -85,B 0,C 180,E1 22101.027,E2 22101.027} C_VEL
LIN {X 0,Y 546.618,Z 951.775,A -85,B 0,C 180,E1 22100.352,E2 22100.352} C_VEL
LIN {X 0,Y 543.265,Z 972.42,A -85,B 0,C 180,E1 22099.546,E2 22099.546} C_VEL
LIN {X 0,Y 539.562,Z 992.621,A -85,B 0,C 180,E1 22098.625,E2 22098.625} C_VEL
LIN {X 0,Y 534.968,Z 1015.371,A -85,B 0,C 180,E1 22097.416,E2 22097.416} C_VEL
LIN {X 0,Y 529.364,Z 1040.073,A -85,B 0,C 180,E1 22095.86,E2 22095.86} C_VEL
LIN {X 0,Y 524.638,Z 1059.396,A -85,B 0,C 180,E1 22094.449,E2 22094.449} C_VEL
LIN {X 0,Y 520.012,Z 1077.406,A -85,B 0,C 180,E1 22092.962,E2 22092.962} C_VEL
LIN {X 0,Y 515.191,Z 1095.47,A -85,B 0,C 180,E1 22091.281,E2 22091.281} C_VEL
LIN {X 0,Y 512.232,Z 1106.263,A -85,B 0,C 180,E1 22090.167,E2 22090.167} C_VEL
LIN {X 0,Y 509.898,Z 1111.983,A -85,B 0,C 180,E1 22089.63,E2 22089.63} C_VEL
LIN {X 0,Y 500.562,Z 1127.214,A -85,B 0,C 180,E1 22088.334,E2 22088.334} C_VEL
LIN {X 0,Y 498.603,Z 1131.683,A -85,B 0,C 180,E1 22087.817,E2 22087.817} C_VEL
LIN {X 0,Y 493.961,Z 1147.44,A -85,B 0,C 180,E1 22085.651,E2 22085.651} C_VEL
LIN {X 0,Y 490.015,Z 1161.005,A -85,B 0,C 180,E1 22083.563,E2 22083.563} C_VEL
LIN {X 0,Y 486.38,Z 1173.955,A -85,B 0,C 180,E1 22081.331,E2 22081.331} C_VEL
LIN {X 0,Y 482.755,Z 1187.468,A -85,B 0,C 180,E1 22078.711,E2 22078.711} C_VEL
LIN {X 0,Y 479.256,Z 1201.391,A -85,B 0,C 180,E1 22075.579,E2 22075.579} C_VEL
LIN {X 0,Y 476.947,Z 1211.523,A -85,B 0,C 180,E1 22072.943,E2 22072.943} C_VEL
LIN {X 0,Y 475.276,Z 1219.97,A -85,B 0,C 180,E1 22070.433,E2 22070.433} C_VEL
LIN {X 0,Y 473.95,Z 1227.655,A -85,B 0,C 180,E1 22067.806,E2 22067.806} C_VEL
LIN {X 0,Y 472.933,Z 1235.078,A -85,B 0,C 180,E1 22064.816,E2 22064.816} C_VEL
LIN {X 0,Y 472.304,Z 1241.786,A -85,B 0,C 180,E1 22061.472,E2 22061.472} C_VEL
LIN {X 0,Y 472.049,Z 1246.131,A -85,B 0,C 180,E1 22058.644,E2 22058.644} C_VEL
LIN {X 0,Y 471.95,Z 1249.034,A -85,B 0,C 180,E1 22056.075,E2 22056.075} C_VEL
LIN {X 0,Y 471.914,Z 1250.854,A -85,B 0,C 180,E1 22053.639,E2 22053.639} C_VEL
LIN {X 0,Y 471.892,Z 1251.772,A -85,B 0,C 180,E1 22051.209,E2 22051.209} C_VEL
LIN {X 0,Y 471.885,Z 1251.787,A -85,B 0,C 180,E1 22048.78,E2 22048.78} C_VEL
LIN {X 0,Y 471.915,Z 1250.892,A -85,B 0,C 180,E1 22046.337,E2 22046.337} C_VEL
LIN {X 0,Y 471.953,Z 1248.995,A -85,B 0,C 180,E1 22043.792,E2 22043.792} C_VEL
LIN {X 0,Y 472.051,Z 1246.075,A -85,B 0,C 180,E1 22041.223,E2 22041.223} C_VEL
LIN {X 0,Y 472.307,Z 1241.711,A -85,B 0,C 180,E1 22038.393,E2 22038.393} C_VEL
LIN {X 0,Y 472.946,Z 1234.969,A -85,B 0,C 180,E1 22035.048,E2 22035.048} C_VEL
LIN {X 0,Y 473.925,Z 1227.87,A -85,B 0,C 180,E1 22032.182,E2 22032.182} C_VEL
LIN {X 0,Y 475.226,Z 1220.212,A -85,B 0,C 180,E1 22029.553,E2 22029.553} C_VEL
LIN {X 0,Y 476.89,Z 1211.787,A -85,B 0,C 180,E1 22027.042,E2 22027.042} C_VEL
LIN {X 0,Y 479.182,Z 1201.681,A -85,B 0,C 180,E1 22024.405,E2 22024.405} C_VEL
LIN {X 0,Y 482.784,Z 1187.337,A -85,B 0,C 180,E1 22021.173,E2 22021.173} C_VEL
LIN {X 0,Y 486.419,Z 1173.792,A -85,B 0,C 180,E1 22018.549,E2 22018.549} C_VEL
LIN {X 0,Y 490.114,Z 1160.666,A -85,B 0,C 180,E1 22016.291,E2 22016.291} C_VEL
LIN {X 0,Y 494.557,Z 1145.48,A -85,B 0,C 180,E1 22013.971,E2 22013.971} C_VEL
LIN {X 0,Y 500.496,Z 1125.289,A -85,B 0,C 180,E1 22011.291,E2 22011.291} C_VEL
LIN {X 0,Y 505.295,Z 1108.759,A -85,B 0,C 180,E1 22009.377,E2 22009.377} C_VEL
LIN {X 0,Y 509.862,Z 1092.767,A -85,B 0,C 180,E1 22007.724,E2 22007.724} C_VEL
LIN {X 0,Y 514.395,Z 1076.385,A -85,B 0,C 180,E1 22006.208,E2 22006.208} C_VEL
LIN {X 0,Y 519.219,Z 1058.235,A -85,B 0,C 180,E1 22004.712,E2 22004.712} C_VEL
LIN {X 0,Y 525.179,Z 1034.633,A -85,B 0,C 180,E1 22003.018,E2 22003.018} C_VEL
LIN {X 0,Y 530.157,Z 1012.635,A -85,B 0,C 180,E1 22001.677,E2 22001.677} C_VEL
LIN {X 0,Y 534.486,Z 991.743,A -85,B 0,C 180,E1 22000.574,E2 22000.574} C_VEL
LIN {X 0,Y 538.314,Z 971.378,A -85,B 0,C 180,E1 21999.65,E2 21999.65} C_VEL
LIN {X 0,Y 542.028,Z 949.048,A -85,B 0,C 180,E1 21998.791,E2 21998.791} C_VEL
LIN {X 0,Y 545.952,Z 920.553,A -85,B 0,C 180,E1 21997.914,E2 21997.914} C_VEL
LIN {X 0,Y 548.413,Z 897.584,A -85,B 0,C 180,E1 21997.367,E2 21997.367} C_VEL
LIN {X 0,Y 550.182,Z 875.688,A -85,B 0,C 180,E1 21996.964,E2 21996.964} C_VEL
LIN {X 0,Y 560.39,Z 662.965,A -85,B 0,C 180,E1 21993.74,E2 21993.74} C_VEL
LIN {X 0,Y 566.845,Z 533.839,A -85,B 0,C 180,E1 21991.772,E2 21991.772} C_VEL
LIN {X 0,Y 556.591,Z 519.185,A -85,B 0,C 180,E1 21989.635,E2 21989.635} C_VEL
LIN {X 0,Y 546.866,Z 506.005,A -85,B 0,C 180,E1 21987.407,E2 21987.407} C_VEL
LIN {X 0,Y 538.75,Z 495.569,A -85,B 0,C 180,E1 21985.357,E2 21985.357} C_VEL
LIN {X 0,Y 534.378,Z 490.066,A -85,B 0,C 180,E1 21984.162,E2 21984.162} C_VEL
LIN {X 0,Y 530.464,Z 485.169,A -85,B 0,C 180,E1 21983.025,E2 21983.025} C_VEL
LIN {X 0,Y 526.323,Z 480.079,A -85,B 0,C 180,E1 21981.744,E2 21981.744} C_VEL
LIN {X 0,Y 522.416,Z 475.283,A -85,B 0,C 180,E1 21980.445,E2 21980.445} C_VEL
LIN {X 0,Y 517.866,Z 470.065,A -85,B 0,C 180,E1 21978.811,E2 21978.811} C_VEL
LIN {X 0,Y 516.779,Z 468.564,A -85,B 0,C 180,E1 21978.384,E2 21978.384} C_VEL
LIN {X 0,Y 513.286,Z 465.05,A -85,B 0,C 180,E1 21976.99,E2 21976.99} C_VEL
LIN {X 0,Y 511.61,Z 462.494,A -85,B 0,C 180,E1 21976.229,E2 21976.229} C_VEL
LIN {X 0,Y 508.167,Z 459.403,A -85,B 0,C 180,E1 21974.646,E2 21974.646} C_VEL
LIN {X 0,Y 506.266,Z 456.183,A -85,B 0,C 180,E1 21973.593,E2 21973.593} C_VEL
LIN {X 0,Y 502.805,Z 453.681,A -85,B 0,C 180,E1 21971.645,E2 21971.645} C_VEL
LIN {X 0,Y 500.816,Z 450.151,A -85,B 0,C 180,E1 21970.177,E2 21970.177} C_VEL
LIN {X 0,Y 500.295,Z 449.551,A -85,B 0,C 180,E1 21969.781,E2 21969.781} C_VEL
LIN {X 0,Y 496.322,Z 446.734,A -85,B 0,C 180,E1 21966.129,E2 21966.129} C_VEL
LIN {X 0,Y 494.784,Z 442.925,A -85,B 0,C 180,E1 21963.128,E2 21963.128} C_VEL
LIN {X 0,Y 494.853,Z 443.049,A -85,B 0,C 180,E1 21957.105,E2 21957.105} C_VEL
LIN {X 0,Y 496.752,Z 447.266,A -85,B 0,C 180,E1 21953.76,E2 21953.76} C_VEL
LIN {X 0,Y 500.767,Z 449.974,A -85,B 0,C 180,E1 21950.286,E2 21950.286} C_VEL
LIN {X 0,Y 502.817,Z 453.725,A -85,B 0,C 180,E1 21948.762,E2 21948.762} C_VEL
LIN {X 0,Y 506.527,Z 456.598,A -85,B 0,C 180,E1 21946.675,E2 21946.675} C_VEL
LIN {X 0,Y 509.073,Z 460.473,A -85,B 0,C 180,E1 21945.323,E2 21945.323} C_VEL
LIN {X 0,Y 512.049,Z 463.075,A -85,B 0,C 180,E1 21943.989,E2 21943.989} C_VEL
LIN {X 0,Y 514.982,Z 467.103,A -85,B 0,C 180,E1 21942.719,E2 21942.719} C_VEL
LIN {X 0,Y 517.181,Z 469.345,A -85,B 0,C 180,E1 21941.864,E2 21941.864} C_VEL
LIN {X 0,Y 521.381,Z 474.794,A -85,B 0,C 180,E1 21940.303,E2 21940.303} C_VEL
LIN {X 0,Y 525.517,Z 480.144,A -85,B 0,C 180,E1 21938.895,E2 21938.895} C_VEL
LIN {X 0,Y 530.417,Z 486.635,A -85,B 0,C 180,E1 21937.354,E2 21937.354} C_VEL
LIN {X 0,Y 536.973,Z 495.618,A -85,B 0,C 180,E1 21935.465,E2 21935.465} C_VEL
LIN {X 0,Y 545.461,Z 507.574,A -85,B 0,C 180,E1 21933.254,E2 21933.254} C_VEL
LIN {X 0,Y 555.939,Z 523.115,A -85,B 0,C 180,E1 21930.8,E2 21930.8} C_VEL
LIN {X 0,Y 566.937,Z 540.544,A -85,B 0,C 180,E1 21928.471,E2 21928.471} C_VEL
LIN {X 0,Y 556.634,Z 751.597,A -85,B 0,C 180,E1 21925.259,E2 21925.259} C_VEL
LIN {X 0,Y 549.593,Z 899.938,A -85,B 0,C 180,E1 21923.008,E2 21923.008} C_VEL
LIN {X 0,Y 547.296,Z 926.451,A -85,B 0,C 180,E1 21922.509,E2 21922.509} C_VEL
LIN {X 0,Y 543.925,Z 953.543,A -85,B 0,C 180,E1 21921.815,E2 21921.815} C_VEL
LIN {X 0,Y 540.728,Z 974.988,A -85,B 0,C 180,E1 21921.126,E2 21921.126} C_VEL
LIN {X 0,Y 537.187,Z 995.843,A -85,B 0,C 180,E1 21920.324,E2 21920.324} C_VEL
LIN {X 0,Y 533.317,Z 1016.193,A -85,B 0,C 180,E1 21919.407,E2 21919.407} C_VEL
LIN {X 0,Y 528.332,Z 1040.252,A -85,B 0,C 180,E1 21918.138,E2 21918.138} C_VEL
LIN {X 0,Y 522.711,Z 1064.333,A -85,B 0,C 180,E1 21916.628,E2 21916.628} C_VEL
LIN {X 0,Y 517.831,Z 1083.989,A -85,B 0,C 180,E1 21915.207,E2 21915.207} C_VEL
LIN {X 0,Y 513.228,Z 1101.691,A -85,B 0,C 180,E1 21913.763,E2 21913.763} C_VEL
LIN {X 0,Y 508.407,Z 1119.605,A -85,B 0,C 180,E1 21912.121,E2 21912.121} C_VEL
LIN {X 0,Y 502.74,Z 1140.309,A -85,B 0,C 180,E1 21909.976,E2 21909.976} C_VEL
LIN {X 0,Y 497.322,Z 1159.407,A -85,B 0,C 180,E1 21907.681,E2 21907.681} C_VEL
LIN {X 0,Y 492.992,Z 1174.942,A -85,B 0,C 180,E1 21905.579,E2 21905.579} C_VEL
LIN {X 0,Y 489.215,Z 1188.738,A -85,B 0,C 180,E1 21903.498,E2 21903.498} C_VEL
LIN {X 0,Y 485.544,Z 1202.791,A -85,B 0,C 180,E1 21901.128,E2 21901.128} C_VEL
LIN {X 0,Y 481.338,Z 1219.641,A -85,B 0,C 180,E1 21897.87,E2 21897.87} C_VEL
LIN {X 0,Y 478.664,Z 1231.452,A -85,B 0,C 180,E1 21895.227,E2 21895.227} C_VEL
LIN {X 0,Y 476.609,Z 1241.395,A -85,B 0,C 180,E1 21892.711,E2 21892.711} C_VEL
LIN {X 0,Y 474.995,Z 1250.33,A -85,B 0,C 180,E1 21890.139,E2 21890.139} C_VEL
LIN {X 0,Y 473.601,Z 1259.882,A -85,B 0,C 180,E1 21886.944,E2 21886.944} C_VEL
LIN {X 0,Y 472.701,Z 1267.278,A -85,B 0,C 180,E1 21883.834,E2 21883.834} C_VEL
LIN {X 0,Y 472.266,Z 1272.256,A -85,B 0,C 180,E1 21881.237,E2 21881.237} C_VEL
LIN {X 0,Y 472.048,Z 1276.177,A -85,B 0,C 180,E1 21878.655,E2 21878.655} C_VEL
LIN {X 0,Y 471.949,Z 1279.067,A -85,B 0,C 180,E1 21876.086,E2 21876.086} C_VEL
LIN {X 0,Y 471.915,Z 1280.874,A -85,B 0,C 180,E1 21873.65,E2 21873.65} C_VEL
LIN {X 0,Y 471.888,Z 1281.779,A -85,B 0,C 180,E1 21871.22,E2 21871.22} C_VEL
LIN {X 0,Y 471.88,Z 1281.803,A -85,B 0,C 180,E1 21868.913,E2 21868.913} C_VEL
LIN {X 0,Y 471.912,Z 1280.948,A -85,B 0,C 180,E1 21866.483,E2 21866.483} C_VEL
LIN {X 0,Y 471.945,Z 1279.19,A -85,B 0,C 180,E1 21864.047,E2 21864.047} C_VEL
LIN {X 0,Y 472.037,Z 1276.35,A -85,B 0,C 180,E1 21861.479,E2 21861.479} C_VEL
LIN {X 0,Y 472.252,Z 1272.481,A -85,B 0,C 180,E1 21858.898,E2 21858.898} C_VEL
LIN {X 0,Y 472.679,Z 1267.555,A -85,B 0,C 180,E1 21856.302,E2 21856.302} C_VEL
LIN {X 0,Y 473.411,Z 1261.155,A -85,B 0,C 180,E1 21853.566,E2 21853.566} C_VEL
LIN {X 0,Y 474.818,Z 1251.413,A -85,B 0,C 180,E1 21850.189,E2 21850.189} C_VEL
LIN {X 0,Y 476.529,Z 1241.834,A -85,B 0,C 180,E1 21847.405,E2 21847.405} C_VEL
LIN {X 0,Y 478.54,Z 1232.033,A -85,B 0,C 180,E1 21844.91,E2 21844.91} C_VEL
LIN {X 0,Y 481.054,Z 1220.872,A -85,B 0,C 180,E1 21842.394,E2 21842.394} C_VEL
LIN {X 0,Y 484.646,Z 1206.389,A -85,B 0,C 180,E1 21839.509,E2 21839.509} C_VEL
LIN {X 0,Y 488.787,Z 1190.378,A -85,B 0,C 180,E1 21836.763,E2 21836.763} C_VEL
LIN {X 0,Y 492.772,Z 1175.739,A -85,B 0,C 180,E1 21834.535,E2 21834.535} C_VEL
